(* CoDeSys 2.3.6.0 project: oscat13.pro *)
(* Libraries: SysLibRtc.lib 5.10.04 09:37:42, Standard.lib 22.11.04 11:21:12, SYSLIBCALLBACK.LIB 20.4.05 10:04:48, Util.lib 15.6.05 09:51:38 *)

(* PLC configuration (modules and I/O channels)
switch_1 AT %IX21.0 [BOOLOnX_I] Ch_1 Digital input
switch_2 AT %IX21.1 [BOOLOnX_I] Ch_2 Digital input
0750-0501 2 DO 24V DC 0.5A [Type_10_2_Channels] node 1, in %IB1 out %QB1 {INTTypePAAssignment = PLC; INTTypeModule = plugged}
  output_1 AT %QX19.0 [BOOLOnX_Q] Ch_1 Digital output
  output_2 AT %QX19.1 [BOOLOnX_Q] Ch_2 Digital output
0750-0501 2 DO 24V DC 0.5A [Type_10_2_Channels] node 2, in %IB2 out %QB2 {INTTypePAAssignment = PLC; INTTypeModule = plugged}
  output_3 AT %QX19.2 [BOOLOnX_Q] Ch_1 Digital output
  output_4 AT %QX19.3 [BOOLOnX_Q] Ch_2 Digital output
0750-0502 2 DO 24V DC 2.0A [Type_10_2_Channels] node 3, in %IB3 out %QB3 {INTTypePAAssignment = PLC; INTTypeModule = plugged}
  aus55 AT %QX19.4 [BOOLOnX_Q] Ch_1 Digital output
  AT %QX19.5 [BOOLOnX_Q] Ch_2 Digital output
0750-0501 2 DO 24V DC 0.5A [Type_10_2_Channels] node 4, in %IB4 out %QB4 {INTTypePAAssignment = PLC; INTTypeModule = plugged}
  heinz AT %QX19.6 [BOOLOnX_Q] Ch_1 Digital output
  AT %QX19.7 [BOOLOnX_Q] Ch_2 Digital output
0750-0523/0010-0000 1DO 230V AC 16A/Relay 1a/Potential free [Type_26_1_Channels] node 5, in %IB5 out %QB5 {INTTypePAAssignment = PLC; INTTypeModule = plugged}
  hand AT %IX21.2 [BOOLOnX_I] Diagnostic bit
  output_16A AT %QX19.8 [BOOLOnX_Q] Digital output
0750-0559 4 AO 0-10V DC [Type_14_4_Channels] node 6, in %IB6 out %QB6 {INTTypePAAssignment = PLC; INTTypeModule = plugged}
  AT %QW0 [WORDOnW_Q] Ch_1 Analog output
  AT %QW1 [WORDOnW_Q] Ch_2 Analog output
  AT %QW2 [WORDOnW_Q] Ch_3 Analog output
  AT %QW3 [WORDOnW_Q] Ch_4 Analog output
0750-0402 4 DI 24 V DC 3.0ms [Type_1_4_Channels] node 7, in %IB7 out %QB7 {INTTypePAAssignment = PLC; INTTypeModule = plugged}
  switch_3 AT %IX21.4 [BOOLOnX_I] Ch_1 Digital input
  switch_4 AT %IX21.5 [BOOLOnX_I] Ch_2 Digital input
  AT %IX21.6 [BOOLOnX_I] Ch_3 Digital input
  AT %IX21.7 [BOOLOnX_I] Ch_4 Digital input
0750-0402 4 DI 24 V DC 3.0ms [Type_1_4_Channels] node 8, in %IB8 out %QB8 {INTTypePAAssignment = PLC; INTTypeModule = plugged}
  AT %IX21.8 [BOOLOnX_I] Ch_1 Digital input
  AT %IX21.9 [BOOLOnX_I] Ch_2 Digital input
  AT %IX21.10 [BOOLOnX_I] Ch_3 Digital input
  AT %IX21.11 [BOOLOnX_I] Ch_4 Digital input
  AT %IX21.12 [BOOLOnX_I] Ch_1 Digital input
  AT %IX21.13 [BOOLOnX_I] Ch_2 Digital input
  AT %IX21.14 [BOOLOnX_I] Ch_3 Digital input
  AT %IX21.15 [BOOLOnX_I] Ch_4 Digital input
dcf77in AT %IX22.0 [BOOLOnX_I] Ch_1 Digital input
dcf77_2 AT %IX22.1 [BOOLOnX_I] Ch_2 Digital input
AT %IX22.2 [BOOLOnX_I] Ch_3 Digital input
AT %IX22.3 [BOOLOnX_I] Ch_4 Digital input
AT %IX22.4 [BOOLOnX_I] Ch_5 Digital input
AT %IX22.5 [BOOLOnX_I] Ch_6 Digital input
AT %IX22.6 [BOOLOnX_I] Ch_7 Digital input
AT %IX22.7 [BOOLOnX_I] Ch_8 Digital input
0750-0431 8 DI 24 V DC 0.2ms [Type_1_8_Channels] node 11, in %IB11 out %QB11 {INTTypePAAssignment = PLC; INTTypeModule = plugged}
  clkin AT %IX22.8 [BOOLOnX_I] Ch_1 Digital input
  AT %IX22.9 [BOOLOnX_I] Ch_2 Digital input
  AT %IX22.10 [BOOLOnX_I] Ch_3 Digital input
  AT %IX22.11 [BOOLOnX_I] Ch_4 Digital input
  AT %IX22.12 [BOOLOnX_I] Ch_5 Digital input
  AT %IX22.13 [BOOLOnX_I] Ch_6 Digital input
  AT %IX22.14 [BOOLOnX_I] Ch_7 Digital input
  AT %IX22.15 [BOOLOnX_I] Ch_8 Digital input
0750-0402 4 DI 24 V DC 3.0ms [Type_1_4_Channels] node 12, in %IB12 out %QB12 {INTTypePAAssignment = PLC; INTTypeModule = plugged}
  AT %IX23.0 [BOOLOnX_I] Ch_1 Digital input
  AT %IX23.1 [BOOLOnX_I] Ch_2 Digital input
  AT %IX23.2 [BOOLOnX_I] Ch_3 Digital input
  AT %IX23.3 [BOOLOnX_I] Ch_4 Digital input
0750-0531 4 DO 24V DC 0.5A [Type_10_4_Channels] node 13, in %IB13 out %QB13 {INTTypePAAssignment = PLC; INTTypeModule = plugged}
  AT %QX19.10 [BOOLOnX_Q] Ch_1 Digital output
  AT %QX19.11 [BOOLOnX_Q] Ch_2 Digital output
  AT %QX19.12 [BOOLOnX_Q] Ch_3 Digital output
  AT %QX19.13 [BOOLOnX_Q] Ch_4 Digital output
0750-0531 4 DO 24V DC 0.5A [Type_10_4_Channels] node 14, in %IB14 out %QB14 {INTTypePAAssignment = PLC; INTTypeModule = plugged}
  AT %QX19.14 [BOOLOnX_Q] Ch_1 Digital output
  AT %QX19.15 [BOOLOnX_Q] Ch_2 Digital output
  AT %QX20.0 [BOOLOnX_Q] Ch_3 Digital output
  AT %QX20.1 [BOOLOnX_Q] Ch_4 Digital output
0750-0531 4 DO 24V DC 0.5A [Type_10_4_Channels] node 15, in %IB15 out %QB15 {INTTypePAAssignment = PLC; INTTypeModule = plugged}
  AT %QX20.2 [BOOLOnX_Q] Ch_1 Digital output
  AT %QX20.3 [BOOLOnX_Q] Ch_2 Digital output
  AT %QX20.4 [BOOLOnX_Q] Ch_3 Digital output
  AT %QX20.5 [BOOLOnX_Q] Ch_4 Digital output
0750-0531 4 DO 24V DC 0.5A [Type_10_4_Channels] node 16, in %IB16 out %QB16 {INTTypePAAssignment = PLC; INTTypeModule = plugged}
  AT %QX20.6 [BOOLOnX_Q] Ch_1 Digital output
  AT %QX20.7 [BOOLOnX_Q] Ch_2 Digital output
  AT %QX20.8 [BOOLOnX_Q] Ch_3 Digital output
  AT %QX20.9 [BOOLOnX_Q] Ch_4 Digital output
0750-0504 4 DO 24V DC 0.5A [Type_10_4_Channels] node 17, in %IB17 out %QB17 {INTTypePAAssignment = PLC; INTTypeModule = plugged}
  AT %QX20.10 [BOOLOnX_Q] Ch_1 Digital output
  AT %QX20.11 [BOOLOnX_Q] Ch_2 Digital output
  AT %QX20.12 [BOOLOnX_Q] Ch_3 Digital output
  AT %QX20.13 [BOOLOnX_Q] Ch_4 Digital output
0750-0550 2 AO 0-10V DC [Type_14_2_Channels] node 18, in %IB18 out %QB18 {INTTypePAAssignment = PLC; INTTypeModule = plugged}
  aout1 AT %QW4 [WORDOnW_Q] Ch_1 Analog output
  AT %QW5 [WORDOnW_Q] Ch_2 Analog output
0750-0556 2 AO ±10V [Type_14_2_Channels] node 19, in %IB19 out %QB19 {INTTypePAAssignment = PLC; INTTypeModule = plugged}
  AT %QW6 [WORDOnW_Q] Ch_1 Analog output
  AT %QW7 [WORDOnW_Q] Ch_2 Analog output
0750-0654 DataExchange Module [Type_23_1_Channels] node 20, in %IB20 out %QB20 {INTTypePAAssignment = PLC; INTTypeModule = plugged}
  AT %IX0.0 [BOOLOnX_I] Parity error or wrong data in a frame
  AT %IX0.1 [BOOLOnX_I] Buffer overflow
  AT %IX0.2 [BOOLOnX_I] Checksum error
  AT %IX0.3 [BOOLOnX_I] receiver timeout
  AT %IX0.4 [BOOLOnX_I] Module timeout
  AT %IB1 [BYTEOnB_I] Input data Byte 0
  AT %IB2 [BYTEOnB_I] Input data Byte 1
  AT %IB3 [BYTEOnB_I] Input data Byte 2
  AT %QB17 [BYTEOnB_Q] Output data Byte 0
  AT %QB18 [BYTEOnB_Q] Output data Byte 1
  AT %QB19 [BYTEOnB_Q] Output data Byte 2
0750-0460 4 AI PT100 (RTD) [Type_44_4_Channels] node 21, in %IB21 out %QB21 {INTTypePAAssignment = PLC; INTTypeModule = plugged}
  AT %IW2 [INTOnW_I] Ch_1 signed Input value
  AT %IW3 [INTOnW_I] Ch_2 signed Input value
  AT %IW4 [INTOnW_I] Ch_3 signed Input value
  AT %IW5 [INTOnW_I] Ch_4 signed Input value
0750-0454 2 AI 4-20mA Diff [Type_8_2_Channels] node 22, in %IB22 out %QB22 {INTTypePAAssignment = PLC; INTTypeModule = plugged}
  AT %IW6 [WORDOnW_I] Ch_1 Input word
  AT %IW7 [WORDOnW_I] Ch_2 Input word
  Ain1 AT %IW8 [WORDOnW_I] Ch_1 Input word
  Ain2 AT %IW9 [WORDOnW_I] Ch_2 Input word
0750-0550 2 AO 0-10V DC [Type_14_2_Channels] node 24, in %IB24 out %QB24 {INTTypePAAssignment = PLC; INTTypeModule = plugged}
  AT %QW10 [WORDOnW_Q] Ch_1 Analog output
  AT %QW11 [WORDOnW_Q] Ch_2 Analog output
0750-0650 RS 232 C Interface (9600/8/1/N) [Type_21_1_Channels] node 25, in %IB25 out %QB25 {INTTypePAAssignment = PLC; INTTypeModule = plugged}
  AT %IX10.0 [BOOLOnX_I] Transmission acknowledgement
  AT %IX10.1 [BOOLOnX_I] Reception request
  AT %IX10.2 [BOOLOnX_I] Initialization acknowledgement
  AT %IX10.3 [BOOLOnX_I] Input buffer is full
  AT %IX10.4 [BOOLOnX_I] Number of received characters Bit 0
  AT %IX10.5 [BOOLOnX_I] Number of received characters Bit 1
  AT %IX10.6 [BOOLOnX_I] Number of received characters Bit 2
  AT %IB21 [BYTEOnB_I] Input data Byte 0
  AT %IB22 [BYTEOnB_I] Input data Byte 1
  AT %IB23 [BYTEOnB_I] Input data Byte 2
  AT %QX12.0 [BOOLOnX_Q] Transmission request
  AT %QX12.1 [BOOLOnX_Q] Reception acknowledgement
  AT %QX12.2 [BOOLOnX_Q] Initialization request
  AT %QX12.4 [BOOLOnX_Q] Number of characters Bit 0
  AT %QX12.5 [BOOLOnX_Q] Number of characters Bit 1
  AT %QX12.6 [BOOLOnX_Q] Number of characters Bit 2
  AT %QB25 [BYTEOnB_Q] Output data Byte 0
  AT %QB26 [BYTEOnB_Q] Output data Byte 1
  AT %QB27 [BYTEOnB_Q] Output data Byte 2
0750-0641 DALI/DSI-Master [Type_36_1_Channels] node 26, in %IB26 out %QB26 {INTTypePAAssignment = PLC; INTTypeModule = plugged}
  AT %IX12.0 [BOOLOnX_I] Transmit accepted
  AT %IX12.1 [BOOLOnX_I] Receive request
  AT %IX12.2 [BOOLOnX_I] Init accepted
  AT %IX12.3 [BOOLOnX_I] Actor Error
  AT %IX12.4 [BOOLOnX_I] Frame Error
  AT %IX12.5 [BOOLOnX_I] Bus Error
  AT %IX12.6 [BOOLOnX_I] General Module Error
  AT %IB25 [BYTEOnB_I] DALI Response
  AT %IB26 [BYTEOnB_I] DALI Address
  AT %IB27 [BYTEOnB_I] Message 3
  AT %IB28 [BYTEOnB_I] Message 2
  AT %IB29 [BYTEOnB_I] Message 1
  AT %QX14.0 [BOOLOnX_Q] Transmit request
  AT %QX14.1 [BOOLOnX_Q] Receive accepted
  AT %QX14.2 [BOOLOnX_Q] Init request
  AT %QB29 [BYTEOnB_Q] DALI Command, DSI dimming value
  AT %QB30 [BYTEOnB_Q] DALI Address
  AT %QB31 [BYTEOnB_Q] Parameter 2
  AT %QB32 [BYTEOnB_Q] Parameter 1
  AT %QB33 [BYTEOnB_Q] Command extension
0750-0460 4 AI PT100 (RTD) [Type_44_4_Channels] node 27, in %IB27 out %QB27 {INTTypePAAssignment = PLC; INTTypeModule = plugged}
  AT %IW15 [INTOnW_I] Ch_1 signed Input value
  AT %IW16 [INTOnW_I] Ch_2 signed Input value
  AT %IW17 [INTOnW_I] Ch_3 signed Input value
  AT %IW18 [INTOnW_I] Ch_4 signed Input value
0750-0642 EnOcean/RF-Receiver [Type_37_1_Channels] node 28, in %IB28 out %QB28 {INTTypePAAssignment = PLC; INTTypeModule = plugged}
  AT %IX19.0 [BOOLOnX_I] Transmission acknowledgement
  AT %IX19.1 [BOOLOnX_I] Reception request
  AT %IX19.2 [BOOLOnX_I] Initialization acknowledgement
  AT %IX19.3 [BOOLOnX_I] Number of received characters Bit 0
  AT %IX19.4 [BOOLOnX_I] Number of received characters Bit 1
  AT %IX19.5 [BOOLOnX_I] Number of received characters Bit 2
  AT %IX19.6 [BOOLOnX_I] Input buffer is full
  AT %IB39 [BYTEOnB_I] Input data Byte 0
  AT %IB40 [BYTEOnB_I] Input data Byte 1
  AT %IB41 [BYTEOnB_I] Input data Byte 2
  AT %QX17.0 [BOOLOnX_Q] Transmission request
  AT %QX17.1 [BOOLOnX_Q] Reception acknowledgement
  AT %QX17.2 [BOOLOnX_Q] Initialization request
0750-0517 2 DO 230V AC 1.0A Rel 2CO (PotFree) [Type_10_2_Channels] node 29, in %IB29 out %QB29 {INTTypePAAssignment = PLC; INTTypeModule = plugged}
  AT %QX20.14 [BOOLOnX_Q] Ch_1 Digital output
  AT %QX20.15 [BOOLOnX_Q] Ch_2 Digital output
0750-0517 2 DO 230V AC 1.0A Rel 2CO (PotFree) [Type_10_2_Channels] node 30, in %IB30 out %QB30 {INTTypePAAssignment = PLC; INTTypeModule = plugged}
  AT %QX21.0 [BOOLOnX_Q] Ch_1 Digital output
  AT %QX21.1 [BOOLOnX_Q] Ch_2 Digital output
win_o AT %IX256.0 [BOOLOnX_I] BOOL
wout_i AT %QX256.0 [BOOLOnX_Q] BOOL
*)

(* Global variable list: Constants *)
VAR_GLOBAL CONSTANT
	PI : REAL := 3.14159265358979323846264338327950288;
	PI2 : REAL := 6.283185307;
	e : REAL := 2.71828182845904523536028747135266249;
END_VAR

VAR_GLOBAL
	ontime: TIME;
END_VAR

(* Global variable list: Globale_Variablen *)
VAR_GLOBAL

	(* 	time and date variables		*)
	gmt : DT;						(*	world time				*)
	DST_enable : BOOL;					(* 	daylight saving time active	*)
	localtime : DT;				(*	current local time			*)
	sun_offset : TIME;				(*	offset of astrological midday in hours when sun stand at south direction	*)
	sun_rise : TOD;				(*	sun rise for current day in local time *)
	sun_set : TOD;				(*	sun set for current day in local time *)
	sun_declination : REAL;		(*	sun angle at midday	*)

	(*	environmental data			*)
	external_temperature : REAL;	(*	outside temperature in °C	*)
	wind_speed : REAL;			(*	wind speed in km/h			*)

END_VAR

(* Global variable list: Setup_Data *)
VAR_GLOBAL RETAIN

(*	geographical position		*)
	latitude : REAL;		(*	geographical position in degrees north of equator			*)
	longitude : REAL;		(*	geographical position in degrees east of prime meridian		*)
	elevation : REAL;		(*	elevation												*)

(*	time zone data			*)
	Time_zone_offset : TIME;		(*	local time zone offset		*)

END_VAR

(* POU mathematical/array functions/_array_init, ST *)
FUNCTION _array_init : REAL
VAR_INPUT
	pt : POINTER TO ARRAY[0..32000] OF REAL;
	size : INT;
	init : REAL;
END_VAR
VAR
	i: INT;
	stop: INT;
END_VAR


(*
version 1.0	2 oct 2006
programmer 	hugo
tested by		tobias

this function will initialize a given array with a value init.
the function needs to be called:	_array_init(adr("array"),sizeof("array"));
this function will manipulate a given array.
the function will not return anything, it will instead manipulate the original array.
because this function works with pointers its very time efficient and it needs no extra memory.

*)
stop := (size - SIZEOF(pt)) / SIZEOF(pt);
FOR i := 0 TO stop DO
	pt^[i] := init;
END_FOR;
END_FUNCTION

(* POU mathematical/array functions/_array_median, ST *)
FUNCTION _array_median : REAL
VAR_INPUT
	pt : POINTER TO ARRAY[0..32000] OF REAL;
	size : INT;
END_VAR
VAR
	i: INT;
	m: INT;
	temp : REAL;
	stop: INT;
END_VAR

(*
version 1.0	2 oct 2006
programmer 	hugo
tested by		tobias

this function will calculate the median of a given array.
in order to do so the ariginal array is sorted and stays sorted after the function finishes
the function needs to be called:	_array_median(adr("array"),sizeof("array"));
this function will manipulate a given array.
the function will return the median of the original array.
for example [12,0,4,7,1] the median is 4 and the array after the function is called is [0,1,4,7,12]
because this function works with pointers its very time efficient and it needs no extra memory.

*)
stop := (size - SIZEOF(pt)) / SIZEOF(pt);
FOR i := 0 TO stop - 1 DO
	FOR m := i + 1 TO stop DO
		IF pt^[i] > pt^[m] THEN
			temp := pt^[i];
			pt^[i] := pt^[m];
			pt^[m] := temp;
		END_IF;
	END_FOR;
END_FOR;
IF even(stop) THEN
	_array_median := pt^[stop/2];
ELSE
	i := TRUNC(stop/2);
	_array_median := (pt^[i] + pt^[i+1])/2;
END_IF;
END_FUNCTION

(* POU mathematical/even, ST *)
FUNCTION even : BOOL
VAR_INPUT
	in : INT;
END_VAR
VAR
	test: INT;
END_VAR


(*
version 1.0	1 oct 2006
programmer 	hugo
tested by		tobias

this function chacks an input for even  value
the output is true if the input is even.
execution time on wago 750 - 841 =  10  us
*)
IF (in MOD 2) = 0 THEN  even := TRUE; ELSE even := FALSE; END_IF;
END_FUNCTION

(* POU mathematical/array functions/_array_sort, ST *)
FUNCTION _array_sort : BOOL
VAR_INPUT
	pt : POINTER TO ARRAY[0..32000] OF REAL;
	size : INT;
END_VAR
VAR
	i: INT;
	m: INT;
	temp : REAL;
	stop: INT;
END_VAR

(*
version 1.0	2 oct 2006
programmer 	hugo
tested by		tobias

this function will sort a given array.
the function needs to be called:	_array_sort(adr("array"),sizeof("array"));
this function will manipulate a given array.
the function will not return anything, it will instead manipulate the original array.
because this function works with pointers its very time efficient and it needs no extra memory.

*)
stop := (size - SIZEOF(pt)) / SIZEOF(pt);
FOR i := 0 TO stop - 1 DO
	FOR m := i + 1 TO stop DO
		IF pt^[i] > pt^[m] THEN
			temp := pt^[i];
			pt^[i] := pt^[m];
			pt^[m] := temp;
		END_IF;
	END_FOR;
END_FOR;
_array_sort := FALSE;
END_FUNCTION

(* POU Building/HLK/actuator_2P, ST *)
FUNCTION_BLOCK actuator_2P
VAR_INPUT
	val : REAL;
	force : BOOL;
	force_in : BOOL;
END_VAR
VAR_INPUT CONSTANT
	self_act_time : TIME := t#10d;
	self_act_cycles : INT := 5;
	cycle_time : TIME := t#10m;
	min_ontime : TIME := t#10s;
	min_offtime : TIME := t#10s;
END_VAR
VAR_OUTPUT
	out :BOOL;
	pos : REAL;
END_VAR
VAR
	last_activation : TIME;
	time_overflow : BOOL;
	count : INT;
	TON : TIME;
END_VAR


(*
version 1.1	7 oct 2006
programmer 	hugo
tested by		tobias

this is an intelligent actuator interface for any 2point actuator like coil drive.
the 2Point actuator can only switch on/off and therefore a input must be converted to on/off cycles.
the interface can be programmed with double click on the symbol for duty cyle, min_ontime and min_offtime to avoid flickering of the valve or flap.
in addition a self_act_time and self_act_cycles ca be programmed to switch n times on/off every self_act_time to avoid a valve to freeze.
a on and off input can be used to force the valve on or off at all times.
a additional pos output will always indicate the current position of a valve.
the input value must be between 0 and 1.

val		force	force_in	pos	out			
X		0		-			X		duty cycle X
-		1		1			1		1
-		1		0			0		0

*)
(* verify input to be between 0 and 1 *)
IF val <0 THEN val := 0; ELSIF val > 1 THEN val := 1; END_IF;

(* check for min ontime or min offtime and wait if not passed *)
IF (out AND TIME() - last_activation < min_ontime) OR (NOT out AND TIME() - last_activation < min_offtime) THEN RETURN;

(* when force off then shutoff valve *)
ELSIF force AND NOT force_in THEN
	pos := 0;
	out := 0;
	last_activation := TIME();
	count := 0;

(* if force on then turn on valve *)

ELSIF force AND force_in THEN
	pos := 1;
	out := 1;
	last_activation := TIME();
	count := 0;

(* if nothing happened for self_act_time then do self activation cycles *)
ELSIF (TIME() - last_activation >= self_act_time AND count = 0 AND self_act_cycles > 0) OR (count > 0 AND count < self_act_cycles * 2) THEN
	out := NOT out;
	last_activation := TIME();
	count := count + 1;
	RETURN;
ELSIF count > 0 THEN
	count := 0;
ELSE
	ton := multime(cycle_time,val);
	IF ton < min_ontime / 2 THEN ton := t#0s; ELSIF ton < min_ontime THEN ton := min_ontime; END_IF;
	IF ton > cycle_time - min_offtime / 2 THEN ton := cycle_time; ELSIF ton > cycle_time - min_offtime THEN ton := cycle_time - min_offtime; END_IF;
	IF ton = t#0s THEN
		IF out =0 THEN
			pos := 0;
			RETURN;
		ELSE
			out := 0;
			pos := 0;
			last_activation := TIME();
		END_IF;
	ELSIF ton = cycle_time THEN
		IF out = 1 THEN
			pos := 1;
			RETURN;
		ELSE
			out := 1;
			pos := 1;
			last_activation := TIME();
		END_IF;
	END_IF;
	pos := TIME_TO_REAL(ton) / TIME_TO_REAL(cycle_time);
	(* output pulse generation *)
	IF out AND TIME() - last_activation >= ton THEN
		out := 0;
		last_activation := TIME();
	ELSIF NOT out AND TIME() - last_activation >= cycle_time - ton THEN
		out := 1;
		last_activation := TIME();
	END_IF;
END_IF;


(*
revision history:

7.10.2006: changes on and off in the be force and force_in for better usability.
7.10.2006: changed error pos could not reach 1 or 0 under certain conditions due to error in code.

*)
END_FUNCTION_BLOCK

(* POU engineering/measurements/cycle_time, ST *)
FUNCTION_BLOCK cycle_time
VAR_INPUT
	rst : BOOL;
END_VAR
VAR_OUTPUT
	ct_min : TIME := t#0s;
	ct_max : TIME := t#0s;
	ct_last : TIME;
	systime : TIME;
	sysdays : INT;
	cycles : DWORD;
END_VAR
VAR
	last_cycle : TIME;
	tx: TIME;
	init: BOOL;
END_VAR


(*
	version 1.1	12 dec 2006
	programmer 	hugo
	tested BY		hans

this function block measures the cycle time and displays the last, min and max cycle time of the current task.
the resolution is 1ms.
the cycles output is a dword counter which counts the cycles.
a rst pulse on the input will reset all data.


*)
tx :=TIME() - last_cycle;
IF rst THEN
	ct_min := t#0s - t#1ms;
	ct_max := t#0ms;
	cycles := 0;
ELSIF last_cycle > t#0s THEN
	IF tx < ct_min THEN ct_min := tx;
	ELSIF tx > ct_max THEN ct_max := tx;
	END_IF;
	ct_last := tx;
ELSIF ct_min = t#0s THEN
	ct_min := t#0s - t#1ms;
END_IF;
IF init THEN
	systime := systime + tx;
		IF systime >= t#1d THEN
			systime := systime - t#1d;
			sysdays := sysdays + 1;
		END_IF;
END_IF;
init := TRUE;
last_cycle := last_cycle + tx;
cycles := cycles + 1;

(* hm 12.12.2006		rev 1.1

added cycles output, a dword cycle counter.

*)
END_FUNCTION_BLOCK

(* POU Time&Date/multime, ST *)
FUNCTION multime : TIME
VAR_INPUT
	t : TIME;
	M : REAL;
END_VAR
VAR
END_VAR


(*
version 1.0	2 oct 2006
programmer 	hugo
tested by		tobias

multiplies a time by a real number and returns a time
*)
multime := REAL_TO_TIME(TIME_TO_REAL(t)*M);
END_FUNCTION

(* POU Building/HLK/actuator_3P, ST *)
FUNCTION_BLOCK actuator_3P
VAR_INPUT
	in : REAL;
	force : BOOL;
	on : BOOL;
	end_pos : BOOL;
	diag : BOOL;
END_VAR
VAR_INPUT CONSTANT
	min_ontime : TIME := t#10s;
	min_offtime : TIME := t#10s;
	max_runtime : TIME := t#60s;
	auto_diag_time : TIME := t#10d;
	cal_runtime : TIME := t#600s;
	switch_available: BOOL;
END_VAR
VAR_OUTPUT
	out1 : BOOL;
	out2 : BOOL;
	pos : REAL;
	busy : BOOL;
	error : BOOL;
END_VAR
VAR
	val: REAL;
	tx : TIME;
	last_diag: TIME;
	last : TIME;
	runtime_1 : TIME;
	runtime_2 : TIME;
	state : INT;
	force_on : BOOL;
	force_off : BOOL;
	rout: FT_rmp;
	end : R_TRIG;
	cal_timer: TIME;
END_VAR


(*
version 1.1	19 oct 2006
programmer 	hugo
tested by		tobias

actuator_3P is an interface for a 3 point actuator.
a 3P actuator is a motor with 2 directions that drives a valve or flap. the position of the valve or flap is controlled by runtime of the motor foreward or backward.
the available inputs are:
in is a real value which specifies the position of the actuator, 0 = 0% and 1 = 100% any value <0 or > 1 is limited to 0 or 1.
a force input must be low for normal operation and if switched high, the motor can only be controlled for 0% or 100% positions with the on input.
an and pos input is available for a end_pos switch, this switch indicates the valve or flap to be at either 0% or 100%
a diag input can at any time start a diag cycle which turns the motor towards the 0% position, then measures the runtime to 100% and then the runtime to 0%
these runtimes are stored and used for absolute positioning of the motor during normal operation.
a setup constand "auto_diag_time can be used to specify how often the actuator repeates this auto_diag cycla automatically.
at power on a cycle is perfomed automatically.
a 0 for this value means auto diag is never performed.

the outputs ar out1 and out2 for up and down direction of the motor. to avoid flickering the output can be programmed for min_ontime and min_offtime.
a pos outout indicates the absulute position of the actuator during operation and a busy output indicates the actuator is busy.
a error output is initiated when the specified max_runtime is reached by any direction during debug.
also when the up and down direction differs by more then 10% the error output is set.

for absolute positioning accuracy the actuator has a setup variable "cal_runtime" if this is set the actuator measures the total runtime of the motors and when this 
cal_runtime is exceeded it resets the actuator to 0% position and sets the output again to assure absolute accuracy.

autodiag and calibration can be shut off by setting the appropriate values to 0.
a switch_available setup variable specifies if end_pos switches are available.

*)
(* setup *)
tx := TIME() - last;
end(clk := end_pos);

(* init only when first started *)
IF state = 0 THEN
	runtime_1 := max_runtime;
	runtime_2 := max_runtime;
	state := 1;
	rout(KR := 1000 / TIME_TO_REAL(runtime_1), KF := 1000 / TIME_TO_REAL(runtime_1) );
	tx := t#0s;
	last := TIME();
	last_diag := last;
END_IF;

(* check for end_sw and stop if reached *)
IF switch_available AND out1 AND end.Q THEN
	(* upper limit has been reached *)
	out1 := 0;
	rout(rmp := 0, in := 1);
	rout.Rmp := 1;
ELSIF switch_available AND out2 AND end.Q THEN
	(* lower limit has been reached *)
	out2 := 0;
	rout(rmp := 0, in := 0);
	rout.Rmp := 1;
END_IF;

(* check for min_offtime and min_ontime and return if it has not elapsed *)
IF NOT busy AND tx < min_offtime THEN RETURN;
ELSIF busy AND tx < min_ontime THEN RETURN;

(* check for last diag cycle and start diag if auto_diag_time has elapsed *)
ELSIF (tx + last - last_diag > auto_diag_time AND state > 10 AND auto_diag_time > t#0s) OR (diag AND state >= 10) THEN state := 1;

(* check if force pin is high *)
ELSIF force THEN state := 10;

(* check if calibration is necessary *)
ELSIF cal_timer > cal_runtime AND state = 99 AND cal_runtime > t#0s THEN state := 20;
END_IF;

(* state machine for operation *)
CASE state OF

1 :	(* diagnostic start *)
	(* all data is reset and out2 is turned on to make sure we start from top position *)
	last_diag := tx + last;
	diag := 0;
	state := 2;
	pos := 0;
	busy := 1;
	last := tx + last;
	out1 := 0;
	out2 := 1;
	RETURN;

2:	(* wait for max_runtime or end_pos to be reached *)
	IF tx < max_runtime AND NOT end.Q THEN RETURN; END_IF;
	state := 3;
	last := tx + last;
	out1 := 1;
	out2 := 0;
	RETURN;

3: 	(* measure runtime_2 *)
	IF tx < max_runtime AND NOT end.Q THEN RETURN; END_IF;
	state := 4;
	runtime_1 := tx;
	last := tx + last;
	out1 := 0;
	out2 := 1;
	RETURN;

4:	(* measure runtime_1 *)
	IF tx < max_runtime AND NOT end.Q THEN RETURN; END_IF;
	state := 99;
	runtime_2 := tx;
	last := tx + last;
	out2 := 0;
	busy := 0;
	(* reset the output ramp generator to the 0% position as the valve is after diags *)
	rout(rmp := 0, in := 0);
	rout.Rmp := 1;
	cal_timer := t#0s;
	IF differ(TIME_TO_REAL(runtime_1), TIME_TO_REAL(runtime_2), TIME_TO_REAL(max_runtime) * 0.1) THEN error := TRUE;
	ELSIF runtime_1 > multime(max_runtime, 0.9) AND switch_available THEN error := TRUE;
	ELSIF runtime_2 > multime(max_runtime, 0.9) AND switch_available THEN error := TRUE;
	END_IF;
	RETURN;

10: (* force pin is active, outputs are forced on or off by the on pin *)
	IF on AND NOT out2 THEN val := 1;
	ELSIF NOT on AND NOT out1 THEN val := 0;
	END_IF;
	IF NOT force THEN state := 99; END_IF;

20 : (* calibrate to allow for correction of positioning error addig up *)
	cal_timer := t#0s;
	state := 21;
	pos := 0;
	busy := 1;
	last := tx + last;
	out1 := 0;
	out2 := 1;
	RETURN;

21:	(* after end_sw or max_runtime we can be sure to have reached the 0% position *)
	IF tx < max_runtime AND NOT end.Q THEN RETURN; END_IF;
	state := 99;
	out2 := 0;
	busy := 0;
	last := tx + last;
	rout(rmp := 0, in := 0);
	rout.Rmp := 1;
	RETURN;

99: (* normal operation *)
	(* only if input changes for an equivalent of min_ontime then change the output *)
	(* if there is a directional change then wait until last step is finished *)
	IF in < TIME_TO_REAL(min_ontime)/TIME_TO_REAL(max_runtime)/2 THEN val := 0;
	ELSIF in > 1 - TIME_TO_REAL(min_ontime)/TIME_TO_REAL(max_runtime)/2 THEN val := 1;
	ELSIF differ(LIMIT(0,in,1), val, TIME_TO_REAL(min_ontime) / TIME_TO_REAL(max_runtime)) OR in = 0 OR in = 1 THEN
		IF in < val AND NOT out1 THEN val := in;
		ELSIF in > val AND NOT out2 THEN val := in;
		END_IF;
	END_IF;

END_CASE;

(* output ramp generator *)
rout(in := val);
out1 := rout.busy AND rout.UD;
out2 := rout.busy AND NOT rout.UD;
pos := rout.out;

(* set the busy output and if busy goes low, then set the last time in order to check for min_offtime *)
IF NOT busy AND rout.busy THEN
	last := tx + last;
ELSIF busy AND NOT rout.busy THEN
	cal_timer := cal_timer + tx;
	last := tx + last;
END_IF;
busy := rout.busy;



(* revision history

19.10.2006	added security checks for end_switch to avoid overrun of the end_switch, hans

*)
END_FUNCTION_BLOCK

(* POU mathematical/functions/FT_rmp, ST *)
FUNCTION_BLOCK FT_rmp
VAR_INPUT
	Rmp : BOOL := TRUE;
	in : REAL;
	KR : REAL;
	KF : REAL;
END_VAR
VAR_OUTPUT
	out : REAL;
	busy : BOOL;
	UD : BOOL;
END_VAR
VAR
	tx: TIME;
	last: TIME;
END_VAR

(*
	version 1.1	8 oct 2006
	programmer 	oscat
	tested BY		oscat

this ramp function follows an input signal with a linear ramp up or down, the up or down speed can be set with KF and KR.
a K factor of 1 means 1 unit per second on the output. K factors can only be positive and not negative.
a busy output signals the ramp is running or busy false means the in value is present on the output.
a rmp input false means the output follows the input dierctly while a rmp = true means the output follows the input with a ramp.
a updn output signal the directon of the ramp (up or down).

*)
tx := TIME() - last;
IF NOT rmp THEN
	out := in;
	busy := FALSE;
ELSIF out > in AND kf > 0 THEN
	(* ramp down *)
	out := out - TIME_TO_REAL(tx) / 1000 * KF;
	IF out < in THEN out := in; END_IF;
ELSIF out < in AND kr > 0 THEN
	(* ramp up *)
	out := out + TIME_TO_REAL(tx) / 1000 * KR;
	IF out > in THEN out := in; END_IF;
END_IF;

(* set busy and dir flags *)
IF out < in THEN
	busy := TRUE;
	ud := 1;
ELSIF out > in THEN
	busy := TRUE;
	ud := 0;
ELSE
	busy := FALSE;
END_IF;
last := last + tx;


(* revision history:

8.10.2006		added ud output

*)
END_FUNCTION_BLOCK

(* POU mathematical/differ, ST *)
FUNCTION differ : BOOL
VAR_INPUT
	in1 : REAL;
	in2 : REAL;
	X : REAL;
END_VAR
VAR
END_VAR

(*
version 1.0	8 oct 2006
programmer 	hugo
tested by		tobias

this function checks if in1 differs more then x from in2
the output is true if in1 < in2 - x or in1 > in2 + X
*)
differ := in1 < in2 - X OR in1 > in2 + X;
END_FUNCTION

(* POU Building/actuator_pump, ST *)
FUNCTION_BLOCK actuator_pump
VAR_INPUT
	in : BOOL;
	manual : BOOL;
	rst : BOOL := FALSE;
END_VAR
VAR_INPUT CONSTANT
	min_ontime : TIME := t#10s;
	min_offtime : TIME := t#10s;
	run_every : TIME := t#10000m;
END_VAR
VAR_OUTPUT
	pump : BOOL;
	runtime : REAL;
	cycles : REAL;
END_VAR
VAR
	tx : TIME;
	last_change : TIME;
	meter : ontime;
	old_man : BOOL;
END_VAR

(*
	version 1.0	4 dec 2006
	programmer 	oscat
	tested BY		oscat

actuator_pump is a pump interface which cam be controlled by an input in and an input manual.
in or manual high turns the pump output on.
a rst input is used to reset the runtime counters.
when the pump was not active for a time run_every the actuator turns on the pump automatically for min_ontime.
two setup variables min_ontime and min_offtime guarantee a minimum runtime and offtime of the pump.
the units are hours and the output type is real to prevent fromoverfow.

*)
tx := TIME();
IF rst THEN
	rst := FALSE;
	meter(rst := 1);
	meter.rst := 0;
ELSIF manual AND NOT pump AND NOT old_man THEN
	last_change := tx;
	pump := 1;
ELSIF NOT manual AND old_man AND pump AND NOT in THEN
	last_change := tx;
	pump := 0;
ELSIF in AND NOT pump AND tx - last_change >= min_offtime THEN
	last_change := tx;
	pump := 1;
ELSIF pump AND NOT in AND NOT manual AND tx - last_change >= min_ontime THEN
	last_change := tx;
	pump := 0;
ELSIF NOT pump AND tx - last_change >= run_every THEN
	last_change := tx;
	pump := 1;
END_IF;

meter(in := pump);
runtime := meter.ontime;
cycles := meter.cycles;
old_man := manual;
END_FUNCTION_BLOCK

(* POU engineering/measurements/ontime, ST *)
FUNCTION_BLOCK ontime
VAR_INPUT
	in : BOOL;
	rst : BOOL := FALSE;
END_VAR
VAR_OUTPUT RETAIN PERSISTENT
	ontime : REAL;
	last_on : REAL;
	cycles : REAL;
END_VAR
VAR
	tx: TIME;
	last : TIME;
	power : BOOL := FALSE;
	edge : BOOL := 0;
END_VAR

(*
version 1.0	4 aug 2006
programmer 	oscat
tested by		tobias

M_runtime measures the ontime of a signal in hours.
the output is of type real because the time type will overflow within 49 days.
the units are hours.

*)
(* at first we need to determine if the sps was powered off *)

tx := TIME();
IF NOT power THEN
	power := TRUE;
	cycles := cycles +1;
ELSIF rst THEN
	ontime := 0;
	cycles := 0;
	last_on := 0;
ELSIF in THEN
	ontime := ontime + DWORD_TO_REAL( TIME_TO_DWORD(tx - last))/3600000.0;
	last_on := last_on + DWORD_TO_REAL(TIME_TO_DWORD(tx - last))/3600000.0;
	IF in AND NOT edge THEN
		cycles := cycles +1;
		last_on := 0;
	END_IF;
END_IF;
last := tx;
edge := in;
END_FUNCTION_BLOCK

(* POU Building/actuator_UD, ST *)
FUNCTION_BLOCK actuator_UD
VAR_INPUT
	UD : BOOL;
	ON : BOOL;
	TON : TIME;
	TOF : TIME;
	Manual : BOOL := 0;
	Up : BOOL;
	Dn : BOOL;
	off : BOOL := 0;
	YUP_in : BOOL;
	YDN_in : BOOL;
END_VAR

VAR_OUTPUT
	Yup : BOOL;
	Ydn : BOOL;
END_VAR
VAR
	tx : TIME;
	last : TIME;
	init: BOOL;
END_VAR

(*
version 1.0	12 Nov 2006
programmer 	hugo
tested by		tobias

out_ud is a up/dn or Right/left locked output driver.
if can be controlled by automatic inputs UD and ON as well as manual inputs for up and dn.
a security input to shut off at any time is prvided by the off input.
to time set inputs ton and toff specify a minimum on time for outputs and a minimum off time befoore the next output can become active.
the module assures that only one output can be active at any time.
for higher security pls make sure you use hardware locking of the outputs to prevent from defective wiring or outputs.
further security is provided b feedback inputs Yup_in and Ydn_in which are separate inputs for the output signal, if these inputs are not available 
pls connect them directly to Yup and Ydn.
automatic mode can override manual mode by setting the on input high while the manual input is high.

*)
tx := TIME();
IF NOT init THEN
	(* INITIALIZATION AT FIRST CALL *)
	last := tx;
	init := TRUE;
ELSIF off THEN
	(* emergency shut off detected *)
	Yup := FALSE;
	Ydn := FALSE;
	last := tx;
ELSIF ((Yup OR Ydn) AND tx - last < Ton) OR ((NOT Yup AND NOT Ydn) AND tx - last < tof) THEN
	(* WATH FOR MIN TON AND TOF TIME *)
	RETURN;
ELSIF manual AND NOT on THEN
	(* manual operation detected *)
	IF UP AND NOT DN AND NOT OFF THEN
		Ydn := 0;
		IF NOT Ydn_in THEN Yup := 1; END_IF;
		last := tx;
	ELSIF DN AND NOT UP AND NOT OFF THEN
		Yup := 0;
		IF NOT Yup_in THEN Ydn := 1; END_IF;
		last := tx;
	ELSE
		IF YUP OR YDN THEN LAST := tx; END_IF;
		Yup := 0;
		Ydn := 0;
	END_IF;
ELSE
	(* automatic operation *)
	IF Ud AND on AND NOT OFF THEN
		Ydn := 0;
		IF NOT ydn_in THEN Yup := 1; END_IF;
		last := tx;
	ELSIF NOT UD AND on AND NOT OFF THEN
		Yup := 0;
		IF NOT yup_in THEN Ydn := 1; END_IF;
		last := tx;
	ELSE
		IF Yup OR Ydn THEN last := tx; END_IF;
		Yup := 0;
		Ydn := 0;
	END_IF;
END_IF;

(* make sure Yup and Ydn are never on at the same time *)
IF Ydn AND Yup_in THEN Ydn := 0; END_IF;
IF Yup AND Ydn_in THEN Yup := 0; END_IF;
END_FUNCTION_BLOCK

(* POU engineering/signal conditioning/AIN, ST *)
FUNCTION AIN : REAL
VAR_INPUT
	in : DWORD;
END_VAR
VAR_INPUT CONSTANT
	Bits : BYTE;
	sign : BYTE := 255;
	low : REAL := 0;
	high : REAL := 10;
END_VAR
VAR
	temp1 : DWORD;
	temp2 : DWORD;
	sx : BOOL;
END_VAR

(*
version 1.1	18 aug 2006
programmer 	oscat
tested by		tobias

Ain converts signals from A/D converters or other analog sources to an internal real value
the lowest number of bits are extracted from the input word and the sign will be extracted if available separately.
the output signal is then conditioned to range from low to high values for a 0 to max value on the analog inputs:
for example a 15bit input (bits := 12) with sign at bit 15 (0..15) will deliver 0.0 (low value at 0) for an input value of 2#0000_0000_0000
an input value of 2#1111_1111_1111 will deliver 10.0 on the output (high value set to 10).

*) 
(* extract the sign bit *)
IF sign < 32 THEN
	temp1 := SHR(in,sign);
	sx := temp1.0;
ELSE
	sx := FALSE;
END_IF;
temp1 := SHR(16#FFFFFFFF,32-bits);
temp2 := in AND temp1;
AIN := (high - low)*temp2 / temp1 + low;

(* revision history
fixed an error with low value negative and high value 0.
hans
*)
END_FUNCTION

(* POU engineering/signal conditioning/Aout_16, ST *)
FUNCTION AOUT_16 : WORD
VAR_INPUT
	in : REAL;
END_VAR
VAR_INPUT CONSTANT
	Bits : BYTE;
	sign : BYTE := 255;
	low : REAL := 0;
	high : REAL := 10;
END_VAR
VAR
	temp : WORD;
	temp2 : WORD;
END_VAR

(*
version 1.0	4 aug 2006
programmer 	oscat
tested by		tobias

this module conditions an internal real value for a signal output D/A converter.
Aout_16 converts and internal real value to a word for an D/A converter or other output devices.
The input value is converted to a n-bit wide output and a sign bit is set separately as specified.
the outout min value is set for the specified min input value and the max output is set for the max input value.
an input higher or lower then the max or min value will set the respective max or min value or the output.


*) 
IF in < low THEN in := low;
ELSIF in > high THEN in := high;
END_IF;
temp := REAL_TO_WORD((in - low) / (high - low) * (EXPT(2,bits) -1));
IF sign_R(in) AND sign < 16 THEN
	temp := SHL(16#0001,sign) OR temp;
END_IF;
Aout_16 := temp;
END_FUNCTION

(* POU mathematical/sign_R, ST *)
FUNCTION sign_R : BOOL
VAR_INPUT
	in : REAL;
END_VAR
VAR
	X : DWORD;
END_VAR

(*
version 1.0	1 sep 2006
programmer 	hugo
tested by		tobias

this function return true if the real input is negative

*)
x := REAL_TO_DWORD(in);
sign_R := x.31;
END_FUNCTION

(* POU mathematical/array functions/array_avg, ST *)
FUNCTION array_avg : REAL
VAR_INPUT
	pt : POINTER TO ARRAY[0..32000] OF REAL;
	size : INT;
END_VAR
VAR
	i: INT;
	stop: INT;
END_VAR

(*
version 1.0	2 oct 2006
programmer 	hugo
tested by		tobias

this function will calculate the average of a given array.
the function needs to be called:	array_avg(adr("array"),sizeof("array"));
because this function works with pointers its very time efficient and it needs no extra memory.

*)
stop := (size -SIZEOF(pt)) / SIZEOF(pt);
array_avg := pt^[0];
FOR i := 1 TO stop DO
	array_avg := array_avg + pt^[i];
END_FOR;
array_avg := array_avg / (stop + 1);
END_FUNCTION

(* POU mathematical/array functions/array_max, ST *)
FUNCTION array_max : REAL
VAR_INPUT
	pt : POINTER TO ARRAY[0..32000] OF REAL;
	size : INT;
END_VAR
VAR
	i: INT;
	stop: INT;
END_VAR

(*
version 1.0	2 oct 2006
programmer 	hugo
tested by		tobias

this function will calculate the max value of a given array.
the function needs to be called:	array_max(adr("array"),sizeof("array"));
because this function works with pointers its very time efficient and it needs no extra memory.

*)
stop := (size -SIZEOF(pt)) / SIZEOF(pt);
array_max := pt^[0];
FOR i := 1 TO stop DO
	IF pt^[i] > array_max THEN array_max := pt^[i]; END_IF;
END_FOR;
END_FUNCTION

(* POU mathematical/array functions/array_min, ST *)
FUNCTION array_min : REAL
VAR_INPUT
	pt : POINTER TO ARRAY[0..32000] OF REAL;
	size : INT;
END_VAR
VAR
	i: INT;
	stop: INT;
END_VAR

(*
version 1.0	2 oct 2006
programmer 	hugo
tested by		tobias

this function will calculate the min value of a given array.
the function needs to be called:	array_min(adr("array"),sizeof("array"));
because this function works with pointers its very time efficient and it needs no extra memory.

*)
stop := (size - SIZEOF(pt)) / SIZEOF(pt);
array_min := pt^[0];
FOR i := 1 TO stop DO
	IF pt^[i] < array_min THEN array_min := pt^[i]; END_IF;
END_FOR;
END_FUNCTION

(* POU mathematical/array functions/array_spr, ST *)
FUNCTION array_spr : REAL
VAR_INPUT
	pt : POINTER TO ARRAY[0..32000] OF REAL;
	size : INT;
END_VAR
VAR
	i: INT;
	stop: INT;
	array_max : REAL;
	array_min : REAL;
END_VAR

(*
version 1.0	2 oct 2006
programmer 	hugo
tested by		tobias

this function will calculate the spread of a given array.
the function needs to be called:	array_spr(adr("array"),sizeof("array"));
for example: spread of [12,0,4,1,7] is 12 - 0 = 12.
because this function works with pointers its very time efficient and it needs no extra memory.

*)
stop := (size -SIZEOF(pt)) / SIZEOF(pt);
array_min := pt^[0];
array_max := pt^[0];
FOR i := 1 TO stop DO
	IF pt^[i] > array_max THEN array_max := pt^[i];
	ELSIF pt^[i] < array_min THEN array_min := pt^[i];
	END_IF;
END_FOR;
array_spr := array_max - array_min;
END_FUNCTION

(* POU mathematical/array functions/array_sum, ST *)
FUNCTION array_sum : REAL
VAR_INPUT
	pt : POINTER TO ARRAY[0..32000] OF REAL;
	size : INT;
END_VAR
VAR
	i: INT;
	stop: INT;
END_VAR


(*
version 1.0	2 oct 2006
programmer 	hugo
tested by		tobias

this function will calculate the sum of a given array.
the function needs to be called:	array_sum(adr("array"),sizeof("array"));
because this function works with pointers its very time efficient and it needs no extra memory.

*)
stop := (size -SIZEOF(pt)) / SIZEOF(pt);
array_sum := pt^[0];
FOR i := 1 TO stop DO
	array_sum := array_sum + pt^[i];
END_FOR;
END_FUNCTION

(* POU mathematical/array functions/array_trend, ST *)
FUNCTION array_trend : REAL
VAR_INPUT
	pt : POINTER TO ARRAY[0..32000] OF REAL;
	size : INT;
END_VAR
VAR
	i: INT;
	stop: INT;
	x: REAL;
	y : REAL;
END_VAR

(*
version 1.0	2 oct 2006
programmer 	hugo
tested by		tobias

this function will calculate the trend of a given array.
trend will calculate the avg of the first half of the array and then the avg of the second half, trend = avg2 - avg1.
for example:  [0,1,4,5,3,4,6,3] = 4 - 2.5 = 1.5
the function needs to be called:	array_trend(adr("array"),sizeof("array"));
because this function works with pointers its very time efficient and it needs no extra memory.

*)
stop := (size - SIZEOF(pt)) / SIZEOF(pt);
FOR i := 0 TO stop / 2 DO x := x + pt^[i]; END_FOR;
X := x / (TRUNC(stop / 2) + 1);
IF even(stop) THEN
	FOR i := stop / 2 TO stop DO y := y + pt^[i]; END_FOR;
	y := y / (stop / 2 + 1);
ELSE
	FOR i := TRUNC(stop / 2) + 1 TO stop DO y := y + pt^[i]; END_FOR;
	y := y / (TRUNC(stop / 2) + 1);
END_IF;
array_trend := y - x;
END_FUNCTION

(* POU Logic/generators/B_TRIG, ST *)
FUNCTION_BLOCK B_TRIG
VAR_INPUT
	CLK : BOOL;
END_VAR
VAR_OUTPUT
	Q : BOOL := 0;
END_VAR
VAR
	edge : BOOL := 0;
END_VAR

(*
version 1.0	4 aug 2006
programmer 	hugo
tested by		tobias

this block is similar to R_trig and F_trig but it generates a pulse on rising and falling edge.

executioin TIME on wago 750-841 = 5us
*)
Q := clk XOR edge;
edge := CLK;
END_FUNCTION_BLOCK

(* POU Logic/gate logic/Bit_of_Dword, ST *)
FUNCTION Bit_of_Dword : BOOL
VAR_INPUT
	in : DWORD;
	N : BYTE;
END_VAR
VAR
	temp: DWORD;
END_VAR

(*
version 1.0	4 aug 2006
programmer 	hugo
tested by		tobias

this function extracts a single bit from the nth position from right (right is lowest bit) *)
temp := SHR(in,n);
Bit_of_Dword := temp.0;
END_FUNCTION

(* POU Logic/gate logic/Bit_to_Byte, ST *)
FUNCTION Bit_to_Byte : BYTE
VAR_INPUT
	B0:BOOL;
	B1:BOOL;
	B2:BOOL;
	B3:BOOL;
	B4:BOOL;
	B5:BOOL;
	B6:BOOL;
	B7:BOOL;
END_VAR
VAR
	Bx : BYTE;
END_VAR

(*
version 1.0	4 aug 2006
programmer 	hugo
tested by		tobias

this function creates a byte from 8 individual bits

executioin TIME on wago 750-841 = 8 us
*)
BX.0 := B0;
BX.1 := B1;
BX.2 := B2;
BX.3 := B3;
BX.4 := B4;
BX.5 := B5;
BX.6 := B6;
BX.7 := B7;
bit_to_byte := BX;
END_FUNCTION

(* POU Logic/gate logic/Byte_to_Bit, ST *)
FUNCTION_BLOCK Byte_to_Bit
VAR_INPUT
	IN: BYTE;
END_VAR
VAR_OUTPUT
	B0: BOOL;
	B1: BOOL;
	B2: BOOL;
	B3: BOOL;
	B4: BOOL;
	B5: BOOL;
	B6: BOOL;
	B7: BOOL;
END_VAR
VAR
END_VAR

(*
version 1.0	4 aug 2006
programmer 	hugo
tested by		tobias

this Function Block extracts the 8 Bits from a byte

executioin TIME on wago 750-841 = 13us
*)
B0 := IN.0;
B1 := IN.1;
B2 := IN.2;
B3 := IN.3;
B4 := IN.4;
B5 := IN.5;
B6 := IN.6;
B7 := IN.7;
END_FUNCTION_BLOCK

(* POU engineering/conversion/C_to_F, ST *)
FUNCTION C_to_F : REAL
VAR_INPUT
	celsius : REAL;
END_VAR
VAR
END_VAR

(*
version 1.0	4 aug 2006
programmer 	hugo
tested by		tobias

this function converts celsius  to fahrenheit 

executioin TIME on wago 750-841 = 15us
*)
C_to_F := celsius * 1.8 + 32;
END_FUNCTION

(* POU Logic/gate logic/check_parity, ST *)
FUNCTION check_parity : BOOL
VAR_INPUT
	in : DWORD;
	p : BOOL;
END_VAR
VAR
	i: INT;
	cnt: INT := 0;
END_VAR

(*
version 1.0	1 oct 2006
programmer 	hugo
tested by		tobias

this function checks for an even partity for a dword and partity bit.

*)
FOR i := 0 TO 31 DO
	IF in.0 THEN cnt := cnt +1; END_IF;
	in := SHR(in,1);
END_FOR;
check_parity := even(cnt) XOR P;
END_FUNCTION

(* POU Logic/generators/CLK_1ms, ST *)
FUNCTION_BLOCK CLK_1ms
VAR_INPUT
END_VAR
VAR_OUTPUT
	Q : BOOL;
END_VAR
VAR
	CLK : BOOL;
	edge : BOOL := 0;
	stime: DWORD;
END_VAR

(*
clk_gen uses the internal sps time to generate one pulse every 1 ms
every pulse is only valid for one cycle so that a edge trigger is not necessary
clk_gen generates pulses depending on the accuracy of the system clock.

be careful, 1ms clocks will only work on very powerful sps cpu's
wago 750 - 841 will work with pulse width >= 10ms
*)
stime := TIME_TO_DWORD(TIME());
clk := stime.0;
Q := clk XOR edge;
edge := CLK;
END_FUNCTION_BLOCK

(* POU Logic/generators/CLK_2ms, ST *)
FUNCTION_BLOCK CLK_2ms
VAR_INPUT
END_VAR
VAR_OUTPUT
	Q : BOOL;
END_VAR
VAR
	CLK : BOOL;
	edge : BOOL := 0;
	stime: DWORD;
END_VAR

(*
clk_gen uses the internal sps time to generate one pulse every 2 ms
every pulse is only valid for one cycle so that a edge trigger is not necessary
clk_gen generates pulses depending on the accuracy of the system clock.

be careful, 1ms clocks will only work on very powerful sps cpu's
wago 750 - 841 will work with pulse width >= 10ms
*)
stime := TIME_TO_DWORD(TIME());
clk := stime.1;
Q := clk XOR edge;
edge := CLK;
END_FUNCTION_BLOCK

(* POU Logic/generators/CLK_4ms, ST *)
FUNCTION_BLOCK CLK_4ms
VAR_INPUT
END_VAR
VAR_OUTPUT
	Q : BOOL;
END_VAR
VAR
	CLK : BOOL;
	edge : BOOL := 0;
	stime: DWORD;
END_VAR

(*
clk_gen uses the internal sps time to generate one pulse every 4 ms
every pulse is only valid for one cycle so that a edge trigger is not necessary
clk_gen generates pulses depending on the accuracy of the system clock.

be careful, 1ms clocks will only work on very powerful sps cpu's
wago 750 - 841 will work with pulse width >= 10ms
*)
stime := TIME_TO_DWORD(TIME());
clk := stime.2;
Q := clk XOR edge;
edge := CLK;
END_FUNCTION_BLOCK

(* POU Logic/generators/CLK_8ms, ST *)
FUNCTION_BLOCK CLK_8ms
VAR_INPUT
END_VAR
VAR_OUTPUT
	Q : BOOL;
END_VAR
VAR
	CLK : BOOL;
	edge : BOOL := 0;
	stime: DWORD;
END_VAR

(*
clk_gen uses the internal sps time to generate one pulse every 8 ms
every pulse is only valid for one cycle so that a edge trigger is not necessary
clk_gen generates pulses depending on the accuracy of the system clock.

be careful, 1ms clocks will only work on very powerful sps cpu's
wago 750 - 841 will work with pulse width >= 10ms
*)
stime := TIME_TO_DWORD(TIME());
clk := stime.3;
Q := clk XOR edge;
edge := CLK;
END_FUNCTION_BLOCK

(* POU Logic/generators/clk_div, ST *)
FUNCTION_BLOCK clk_div
VAR_INPUT
	clk : BOOL;
	rst: BOOL;
END_VAR
VAR_OUTPUT
	Q0 : BOOL := 0;
	Q1 : BOOL := 0;
	Q2 : BOOL := 0;
	Q3 : BOOL := 0;
	Q4 : BOOL := 0;
	Q5 : BOOL := 0;
	Q6 : BOOL := 0;
	Q7 : BOOL := 0;
END_VAR
VAR
	cnt: BYTE := 0;
END_VAR

(*
version 1.0	4 aug 2006
programmer 	hugo
tested by		tobias

this is a clock divider
each output divides the signal by 2
Q0 = clk / 2 , Q1 = Q0 / 2 and so on.
the outputs have a 50% duty cycle each.


*)
IF clk AND NOT rst THEN
	cnt:= cnt +1;
	Q0 := cnt.0;
	Q1 := cnt.1;
	Q2 := cnt.2;
	Q3 := cnt.3;
	Q4 := cnt.4;
	Q5 := cnt.5;
	Q6 := cnt.6;
	Q7 := cnt.7;
END_IF;
IF rst THEN
	cnt:= 0;
	Q0 := 0;
	Q1 := 0;
	Q2 := 0;
	Q3 := 0;
	Q4 := 0;
	Q5 := 0;
	Q6 := 0;
	Q7 := 0;
END_IF;
END_FUNCTION_BLOCK

(* POU Logic/generators/CLK_Prg, ST *)
FUNCTION_BLOCK CLK_Prg
VAR_INPUT
	PT : TIME := t#10ms;
END_VAR
VAR_OUTPUT
	Q : BOOL := 0;
END_VAR
VAR
	pti : TIME := t#0ms;
	next_pulse: TIME := T#0s;
	run: BOOL := FALSE;
	overflow: BOOL := FALSE;
END_VAR

(*
version 1.0	4 aug 2006
programmer 	hugo
tested by		tobias

clk_prg uses the internal sps time to generate a clock with programmable period time.
the period time is defined for 10ms .. 65s
if the period time is set to less then 10ms the min clock perid is 10ms.
the first cycle after start is a clk pulse and then depending on the programmed period time a delay.
every pulse is only valid for one cycle so that a edge trigger is not necessary
clk_prg depending on the accuracy of the system clock.

*)
IF NOT run THEN
	next_pulse := TIME();
	run := TRUE;
	IF pt < T#10ms THEN PTI := T#10ms; ELSE pti := pt; END_IF;
END_IF;
IF TIME() >= next_pulse AND NOT overflow THEN
	Q := TRUE;
	IF next_pulse + pti < next_pulse THEN
		overflow := TRUE;
	END_IF;
	next_pulse := next_pulse + pti;
ELSE
	Q := FALSE;
	IF TIME() <= next_pulse THEN overflow := FALSE; END_IF;
END_IF;
END_FUNCTION_BLOCK

(* POU Logic/generators/CLK_Pulse, ST *)
FUNCTION_BLOCK CLK_Pulse
VAR_INPUT
	PT : TIME := t#10ms;
	N : INT := 0;
	rst : BOOL := 0;
END_VAR
VAR_OUTPUT
	Q : BOOL := 0;
	cnt : INT := 0;
	run : BOOL := 0;
END_VAR
VAR
	pti : TIME := t#0ms;
	next_pulse: TIME := T#0s;
	overflow: BOOL := FALSE;
END_VAR

(*
version 1.0	4 aug 2006
programmer 	hugo
tested by		tobias

clk_pulse uses the internal sps time to generate a clock with programmable period time.
the period time is defined for 10ms .. 65s.
pulse generation is continuous if N = 0 and for n pulses otherwise.
if the period time is set to less then 10ms the min clock perid is 10ms.
the first cycle after start is a clk pulse and then depending on the programmed period time a delay.
every pulse is only valid for one cycle so that a edge trigger is not necessary
clk_prg depending on the accuracy of the system clock.

*)
IF rst THEN
	run := FALSE;
	pti := t#0ms;
	next_pulse := t#0ms;
	overflow := FALSE;
	Q := FALSE;
	cnt := 0;
ELSIF cnt <= N OR N = 0 THEN
	IF NOT run THEN
		next_pulse := TIME();
		run := TRUE;
		IF pt < T#10ms THEN PTI := T#10ms; ELSE pti := pt; END_IF;
	END_IF;
	IF TIME() >= next_pulse AND NOT overflow AND (cnt < N OR N = 0) THEN
		Q := TRUE;
		cnt := cnt + 1;
		IF next_pulse + pti < next_pulse THEN
			overflow := TRUE;
		END_IF;
		next_pulse := next_pulse + pti;
	ELSE
		Q := FALSE;
		IF cnt = N THEN run := FALSE; END_IF
		IF TIME() <= next_pulse THEN overflow := FALSE; END_IF;
	END_IF;
END_IF
END_FUNCTION_BLOCK

(* POU Time&Date/day_of_month, ST *)
FUNCTION day_of_month : INT
VAR_INPUT
	idate : DATE;
END_VAR
VAR
	yd: INT;
	day_in_year: DWORD;
	day_in_year_begin: DWORD;
	yr: INT;
END_VAR

(*
version 1.0	4 aug 2006
programmer 	hugo
tested by		tobias

returns the day OF month from any DATE
execution TIME with wago 750-841 = 65 us
*)
yr := DWORD_TO_INT((DATE_TO_DWORD(idate)/864+71954300)/36525);
yd := DWORD_TO_INT(DATE_TO_DWORD(idate)/86400 - TRUNC((yr-1)*365.25) + 719178);
IF yr MOD 4 = 0 THEN
	CASE yd OF
		1..31 	:	day_of_month := yd;
		32..60	:	day_of_month := yd - 31;
		61..91	:	day_of_month := yd - 60;
		92..121 :	day_of_month := yd - 91;
		122..152:	day_of_month := yd - 121;
		153..182:	day_of_month := yd - 152;
		183..213:	day_of_month := yd - 182;
		214..244:	day_of_month := yd - 213;
		245..274:	day_of_month := yd - 244;
		275..305:	day_of_month := yd - 274;
		306..335:	day_of_month := yd - 305;
		336..366:	day_of_month := yd - 335;
	END_CASE;
	ELSE
	CASE yd OF
		1..31 	:	day_of_month := yd;
		32..59	:	day_of_month := yd - 31;
		60..90	:	day_of_month := yd - 59;
		91..120 :	day_of_month := yd - 90;
		121..151:	day_of_month := yd - 120;
		152..181:	day_of_month := yd - 151;
		182..212:	day_of_month := yd - 181;
		213..243:	day_of_month := yd - 212;
		244..273:	day_of_month := yd - 243;
		274..304:	day_of_month := yd - 273;
		305..334:	day_of_month := yd - 304;
		335..365:	day_of_month := yd - 334;
	END_CASE;
	END_IF;




(*
this function is simple but took too long with 133 us
the problem is date_to_string is far too slow
day_of_month := STRING_TO_INT(RIGHT(DATE_TO_STRING(idate),2));
*)
END_FUNCTION

(* POU Time&Date/day_of_year, ST *)
FUNCTION day_of_year : INT
VAR_INPUT
	idate : DATE;
END_VAR
VAR
END_VAR

(*
version 1.0	4 aug 2006
programmer 	hugo
tested by		tobias

calculates the day of the year 
execution time for wago 750-841 = 44 us  
*)
day_of_year := DWORD_TO_INT(DATE_TO_DWORD(idate)/86400 + 719178 - TRUNC((year(idate)-1)*365.25));
END_FUNCTION

(* POU Time&Date/year, ST *)
FUNCTION year : INT
VAR_INPUT
	idate : DATE;
END_VAR
VAR
END_VAR

(*
version 1.0	4 aug 2006
programmer 	hugo
tested by		tobias

returs the year of a date  
the function works for dates from 1970 - 2099 
execution time on wago 750-841 = 20us   
*)
year := DWORD_TO_INT((DATE_TO_DWORD(idate)/864+71954300)/36525);
END_FUNCTION

(* POU Time&Date/day_to_time, ST *)
FUNCTION day_to_time : TIME
VAR_INPUT
	input : REAL;
END_VAR
VAR
END_VAR

(*
version 1.0	4 aug 2006
programmer 	hugo
tested by		tobias

converts an amount of days in real to time 
execution time on wago 750-841 =  17 us 
*)
day_to_time := DWORD_TO_TIME(REAL_TO_DWORD(input * 86400000));
END_FUNCTION

(* POU Time&Date/DCF77, ST *)
FUNCTION_BLOCK DCF77
VAR_INPUT
	rec : BOOL;
END_VAR
VAR_INPUT CONSTANT
	sync_timeout : TIME := t#2m;
	time_offset : TIME := t#1h;
	dst_en : BOOL := TRUE;
END_VAR
VAR_OUTPUT
	TP : BOOL;
	DST : BOOL;
	weekday : INT;
	error: BOOL := TRUE;
	RTC : DT;
	RTC1 : DT;
	msec : INT;
	sync : BOOL;
END_VAR
VAR
	MEZ : DT;
	UTC : DT;
	state : INT;
	edge: BOOL;
	tx : TIME;
	ty: TIME;
	last : TIME;
	bits : ARRAY[0..58] OF BOOL;
	cnt : INT;
	i : INT;
	old_time : DT;
	minute : INT;
	hour : INT;
	day : INT;
	month : INT;
	year : INT;
	last_sync: TIME;
END_VAR


(*
version 1.0	2 oct 2006
programmer 	hugo
tested by		tobias

this is a decoder for a DCF77 signal.
the decoder decodes the DCF77 signal and checks for a valid Date_Time.
since the dcf77 signal is only secured with a simple parity the decoder waits for two consecutive valid transmissions before it sets the output signals.
given a valid reception by the receiver the decoder can take up to 3 minutes to start its clocks the first time.
after a valid signal is detected the error output goes low and dignals a valid dcf signal from the receiver.
a tp is only valid for one program cycle to allow for external rtc setting.
after a valid signal is detected two independent internal clocks are started (RTC and RTC1), the seconds  of these clocks are generated by software since the dcf signal is only valid for minutes.
rtc is always utc ( world time) and rtc1 can be set to any time zone by setting the time_zone_offset and enabling dst for automatic summertime.
a sync output signals the the rtc and rtc1 are in sync with the dcf77 signal, if the dcf77 signal is lost for more then the sync time the sync output goes low
but the rtc and rtc1 outputs keep running based on software timing until a valid dcf77 signal is received again and triggers the clock.
in addition a millisecond output gives further resolutionof the clocks.
a dst output shows if daylight saving time is enables and the weekday output shows which day of week currently is ( 1= monday ... 7= sunday).


*)
(* if tp was set it should only be active for 1 cycle *)
TP := FALSE;
IF rec XOR edge THEN
	tx := TIME() - last;
	edge := rec;
	IF NOT rec AND tx > t#1700ms AND tx < t#2000ms THEN
		(* start condition reached *)
		state := 0;
		tp := NOT error;
	ELSIF NOT rec AND tx > t#700ms AND tx < t#1000ms THEN
		(* second switch detected *)
		IF state < 58 THEN state := state +1; ELSE state := 0; END_IF;
	ELSIF rec AND tx  < t#120ms THEN
		(* bit 0 detected  *)
		bits[state] := 0;
	ELSIF rec AND tx > t#120ms AND tx < t#250ms THEN
		(* bit 1 detected *)
		bits[state] := 1;
	ELSE
		(* error condition received signal is not valid *)
		error := TRUE;
		state := 0;
	END_IF;
	last := last + tx;
	IF rec AND state = 58 THEN
		error := FALSE;
		(* decode the bits and check for possible errors *)
		IF bits[0] OR NOT (bits[17] XOR bits[18]) OR NOT bits[20] THEN error := TRUE; END_IF;
		(* decode minute *)
		minute := 0;
		minute.0 := bits[21];
		minute.1 := bits[22];
		minute.2 := bits[23];
		minute.3 := bits[24];
		IF bits[25] THEN minute := minute + 10; END_IF;
		IF bits[26] THEN minute := minute +20; END_IF;
		IF bits[27] THEN minute := minute +40; END_IF;
		IF minute > 59 OR (bits[21] XOR bits[22] XOR bits[23] XOR bits[24] XOR bits[25] XOR bits[26] XOR bits[27] XOR bits[28]) THEN error := TRUE; END_IF;

		(* decode hour *)
		hour := 0;
		hour.0 := bits[29];
		hour.1 := bits[30];
		hour.2 := bits[31];
		hour.3 := bits[32];
		IF bits[33] THEN hour := hour + 10; END_IF;
		IF bits[34] THEN hour := hour +20; END_IF;
		IF hour > 23 OR (bits[29] XOR bits[30] XOR bits[31] XOR bits[32] XOR bits[33] XOR bits[34] XOR bits[35]) THEN error := TRUE; END_IF;

		(* decode day of month *)
		day := 0;
		day.0 := bits[36];
		day.1 := bits[37];
		day.2 := bits[38];
		day.3 := bits[39];
		IF bits[40] THEN day := day + 10; END_IF;
		IF bits[41] THEN day := day + 20; END_IF;
		IF day > 31 THEN error := TRUE; END_IF;

		(* decode day of week *)
		weekday := 0;
		weekday.0 := bits[42];
		weekday.1 := bits[43];
		weekday.2 := bits[44];
		IF weekday > 7 OR weekday < 1 THEN error := TRUE; END_IF;

		(* decode month *)
		month := 0;
		month.0 := bits[45];
		month.1 := bits[46];
		month.2 := bits[47];
		month.3 := bits[48];
		IF bits[49] THEN month := month +10; END_IF;
		IF month > 12 THEN error := TRUE; END_IF;

		(* decode year *)
		year := 0;
		year.0 := bits[50];
		year.1 := bits[51];
		year.2 := bits[52];
		year.3 := bits[53];
		IF bits[54] THEN year := year + 10; END_IF;
		IF bits[55] THEN year := year + 20; END_IF;
		IF bits[56] THEN year := year + 40; END_IF;
		IF bits[57] THEN year := year + 80; END_IF;

		(* check parity for bits 36 to 58 *)
		cnt := 0;
		FOR i := 36 TO 58 DO IF bits[i] THEN cnt := cnt + 1; END_IF; END_FOR;
		IF NOT even(cnt) THEN error := TRUE; END_IF;

		(* time must be valid for two cycles to clear error flag *)
		IF NOT error THEN
			(* set outputs *)
			old_time := mez;
			IF year >= 70 THEN year := year + 1900; ELSE year := year + 2000; END_IF;
			mez := set_DT(year,month,day,hour,minute,0);
			DST := bits[17];
			IF DST THEN UTC := mez - t#2h; ELSE utc := mez - t#1h; END_IF;
			(* set trigger signal only if the receiver has received 2 successive minutes *)
			IF mez <> old_time + t#1m THEN error := TRUE ; END_IF;
		END_IF;
	END_IF;
END_IF;

(* this portion implements a free running clock which is triggered by the dcf77 signal *)
IF tp THEN
	rtc := utc;
	IF DST AND dst_en THEN rtc1 := rtc + time_offset + t#1h; ELSE rtc1 := rtc + time_offset; END_IF;
	sync := TRUE;
	last_sync := last;
	ty := last;
ELSIF rtc > DWORD_TO_DT(0) AND TIME() - ty >= t#1s THEN
	rtc := rtc + t#1s;
	rtc1 := rtc1 + t#1s;
	ty := ty + t#1s;
	sync := ty - last_sync < sync_timeout AND last_sync > DWORD_TO_TIME(0);
END_IF;
msec := TIME_TO_INT(TIME() - ty);



(* decode information
bits		content
0			Bitwert immer 0
1 bis 14	reserviert für Betriebsinformationen (nicht für DCF77-Nutzer bestimmt)
15			Rufbit für Alarmierung der PTB-Mitarbeiter
			(bis Mai 2003: Bitwert = 0 falls normale Antenne in Verwendung; 1 = Backupantenne)
16			Bitwert = 1 falls ein Wechsel von MEZ nach MESZ oder umgekehrt bevorsteht; Dauer der Anzeige: 1 Stunde
17 + 18	gültige Zeit = MEZ, falls Bit 17=0 und Bit 18=1
			gültige Zeit = MESZ, falls Bit 17=1 und Bit 18=0
19			Bitwert = 1 falls innerhalb den nächsten 59 Minuten eine Schaltsekunde angeordnet ist. Beim Einfügen einer Schaltsekunde wird anstelle der 59. die 60. Sekundenmarke weggelassen und in der 58. erfolgt ausnahmsweise ein Trägerabfall.
20			Startbit für Zeitinformation (immer 1)
21 - 27		1, 2, 4, 8, 10, 20, 40 Minuten (bitweise Addition)
28			Prüfbit (gerade Parität) für die Bits 21-27
29 - 34		1, 2, 4, 8, 10, 20 Stunden (bitweise Addition)
35			Prüfbit (gerade Parität) für die Bits 29-34
36 - 41		Tagesnummer im aktuellen Monat: 1, 2, 4, 8, 10, 20 (bitweise Addition)
42 - 44		Tagesnummer in der aktuellen Woche: 1, 2, 4 (bitweise Addition)
45 - 49		Monatsnummer: 1, 2, 4, 8, 10 (bitweise Addition)
50 - 57		Jahr (zweistellig): 1, 2, 4, 8, 10, 20, 40, 80 (bitweise Addition)
58			Prüfbit (gerade Parität) füR die Bits 36-57

*)
END_FUNCTION_BLOCK

(* POU Time&Date/DST, ST *)
FUNCTION DST : BOOL
VAR_INPUT
	utc : DT;
	time_zone_offset : TIME;
END_VAR
VAR
	yr : INT;
	yr4 : DWORD;
	ltc: DWORD;
	idate : DWORD;
END_VAR

(*
version 1.0	4 aug 2006
programmer 	hugo
tested by		tobias

 this functions returns TRUE IF dst TIME is active 
 the FUNCTION calculates automaticall FOR any year betweek 1970 AND 2099 
wheather daylight savings is on OR off 
the summertime calculation is done according to european standards.
dst will become TRUE AT 02:00 in the morning FOR the respective days 
AND it will become FALSE after daylight savings TIME is switched back end OF october automatically 
(execution TIME on wago 750-841 =  110us   
*)
yr := year(DT_TO_DATE(utc));
ltc := DT_TO_DWORD(utc+time_zone_offset);
idate := DT_TO_DWORD(set_DT(yr,3,31,2,0,0));
yr4 := 5*yr/4;
IF idate - ((yr4+4) MOD 7)*86400 <= ltc AND idate + (214 - (yr4+1) MOD 7)*86400 > ltc THEN DST := TRUE; ELSE DST := FALSE; END_IF;


(*

Equation used TO calculate the beginning OF European Summer TIME:
Sunday (31 - (5*y/4 + 4) mod 7) March at 01.00 UTC
(valid through 2099, courtesy of Robert H. van Gent, EC).

European Summer Time ends (clocks go back) at 01.00 UTC on

    * 29 October 2006
    * 28 October 2007
    * 26 October 2008

Equation used to calculate the end of European Summer Time:
Sunday (31 - (5*y/4 + 1) mod 7) October at 01.00 UTC
(validity AND credits as above).

*)
END_FUNCTION

(* POU Time&Date/set_DT, ST *)
FUNCTION set_DT : DT
VAR_INPUT
	year : INT;
	month : INT;
	day : INT;
	hour : INT;
	minute : INT;
	second : INT;
END_VAR
VAR
	count : DWORD;
	leap : BOOL;
END_VAR

(*
version 1.0	4 aug 2006
programmer 	hugo
tested by		tobias


creates a date output from year, month and day of month
year must be in the form of 4 digits ie 2006 or 1977.
execution time on wago 750-841 = 45 us   
*)
IF year MOD 4 = 0 THEN leap := TRUE; ELSE leap := FALSE; END_IF;
count := TRUNC((year-1)*365.25-719178+day);
CASE month OF
2:	count := count + 31;
3:	IF leap THEN count := count + 60; ELSE count := count + 59; END_IF;
4:	IF leap THEN count := count + 91; ELSE count := count + 90; END_IF;
5:	IF leap THEN count := count + 121; ELSE count := count + 120; END_IF;
6:	IF leap THEN count := count + 152; ELSE count := count + 151; END_IF;
7:	IF leap THEN count := count + 182; ELSE count := count + 181; END_IF;
8:	IF leap THEN count := count + 213; ELSE count := count + 212; END_IF;
9:	IF leap THEN count := count + 244; ELSE count := count + 243; END_IF;
10:	IF leap THEN count := count + 274; ELSE count := count + 273; END_IF;
11:	IF leap THEN count := count + 305; ELSE count := count + 304; END_IF;
12:	IF leap THEN count := count + 335; ELSE count := count + 334; END_IF;
END_CASE;
set_DT := DWORD_TO_DT(count * 86400 + second + minute * 60 + hour * 3600);
END_FUNCTION

(* POU Time&Date/month, ST *)
FUNCTION month : INT
VAR_INPUT
	idate : DATE;
END_VAR
VAR
END_VAR

(*
version 1.0	4 aug 2006
programmer 	hugo
tested by		tobias

returns the month of a date  
execution time on wago 750-841 = 145us
*)
month := STRING_TO_INT(MID(DATE_TO_STRING(idate),2,8));
END_FUNCTION

(* POU Time&Date/hour, ST *)
FUNCTION hour : INT
VAR_INPUT
	itod : TOD;
END_VAR
VAR
END_VAR

(*
version 1.0	4 aug 2006
programmer 	hugo
tested by		tobias

extracts the hour of a Time_of_day 
execution time for wago 750-841 = 10 us  
*)
hour := DWORD_TO_INT(TOD_TO_DWORD(itod)/3600000);




(* change history

2.10.2006 changes name of input to itod

*)
END_FUNCTION

(* POU Time&Date/minute, ST *)
FUNCTION minute : INT
VAR_INPUT
	itod : TOD;
END_VAR
VAR
END_VAR

(*
version 1.1	2 oct 2006
programmer 	hugo
tested by		tobias

extracts the minutes out of TOD truncating the ceconds 
execution time on wago 750-841  = 18us

*)  
minute := DWORD_TO_INT(TOD_TO_DWORD(itod)/60000 - TOD_TO_DWORD(itod)/3600000 * 60);


(* change history

2.10.2006 changes name of input to itod

*)
END_FUNCTION

(* POU Time&Date/second, ST *)
FUNCTION second : REAL
VAR_INPUT
	itod : TOD;
END_VAR
VAR
END_VAR

(*
version 1.1	2 oct 2006
programmer 	hugo
tested by		tobias

returns the seconds and milliseconds as real of TOD   
execution time on wago 750-841 = 20 us 
*)
second := DWORD_TO_REAL(TOD_TO_DWORD(itod) - TOD_TO_DWORD(itod)/60000 * 60000)/1000;



(* change history

2.10.2006 changes name of input to itod

*)
END_FUNCTION

(* POU Time&Date/weekday, ST *)
FUNCTION weekday : INT
VAR_INPUT
	idate : DATE;
END_VAR
VAR
END_VAR

(*
version 1.1	21 aug 2006
programmer 	hugo
tested by		tobias

calculates the weekday of a week   
monday = 1 ..... sunday = 7  
execution time on wago 750-841 = 22 us  
*)
weekday := DWORD_TO_INT((DATE_TO_DWORD(idate)/86400+3) MOD 7)+1;

(* corrected a miscalculation formula is now correct *)
END_FUNCTION

(* POU Logic/gate logic/DEC_2, CFC *)
FUNCTION_BLOCK DEC_2
VAR_INPUT
	D: BOOL;
	A: BOOL;
END_VAR
VAR_OUTPUT
	Q0: BOOL;
	Q1: BOOL;
END_VAR
VAR
END_VAR

(*
version 1.0	4 aug 2006
programmer 	hugo
tested by		tobias

a bit input will be decoded to the two outputs Q0 or Q1
dependent on the value of A
A=0 decodes to Q0 and A=1 decodes to Q1

executioin TIME on wago 750-841 = 5us
*)
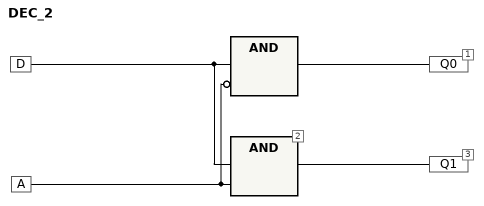
_CFC_ (* Continuous Function Chart, elements in execution order *)
#0 AND(D, NOT A)
#1 Q0 <= #0
#2 AND(D, A)
#3 Q1 <= #2
_END_CFC_
(* the same logic as Structured Text *)
Q0 := D AND NOT A;
Q1 := D AND A;
END_FUNCTION_BLOCK

(* POU Logic/gate logic/DEC_4, CFC *)
FUNCTION_BLOCK DEC_4
VAR_INPUT
	D: BOOL;
	A0: BOOL;
	A1: BOOL;
END_VAR
VAR_OUTPUT
	Q0: BOOL;
	Q1: BOOL;
	Q2: BOOL;
	Q3: BOOL;
END_VAR
VAR
END_VAR

(*
version 1.0	4 aug 2006
programmer 	hugo
tested by		tobias

a bit input will be decoded to one of the 4 outputs
dependent on the Adress on A0 and A1

executioin TIME on wago 750-841 = 9us
*)
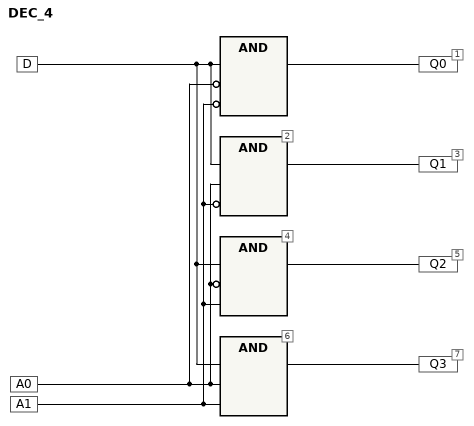
_CFC_ (* Continuous Function Chart, elements in execution order *)
#0 AND(D, NOT A0, NOT A1)
#1 Q0 <= #0
#2 AND(D, A0, NOT A1)
#3 Q1 <= #2
#4 AND(D, NOT A0, A1)
#5 Q2 <= #4
#6 AND(D, A0, A1)
#7 Q3 <= #6
_END_CFC_
(* the same logic as Structured Text *)
Q0 := D AND NOT A0 AND NOT A1;
Q1 := D AND A0 AND NOT A1;
Q2 := D AND NOT A0 AND A1;
Q3 := D AND A0 AND A1;
END_FUNCTION_BLOCK

(* POU Logic/gate logic/DEC_8, CFC *)
FUNCTION_BLOCK DEC_8
VAR_INPUT
	D: BOOL;
	A0: BOOL;
	A1: BOOL;
	A2: BOOL;
END_VAR
VAR_OUTPUT
	Q0: BOOL;
	Q1: BOOL;
	Q2: BOOL;
	Q3: BOOL;
	Q4: BOOL;
	Q5: BOOL;
	Q6: BOOL;
	Q7: BOOL;
END_VAR
VAR
END_VAR

(*
version 1.0	4 aug 2006
programmer 	hugo
tested by		tobias

a bit input will be decoded to one of the 8 outputs
dependent on the Adress on A0, A1 and A2

executioin TIME on wago 750-841 = 17us
*)
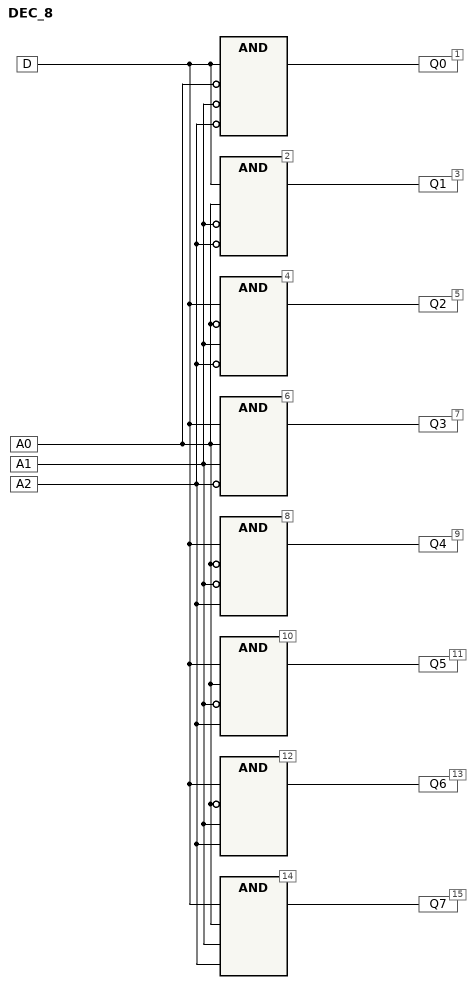
_CFC_ (* Continuous Function Chart, elements in execution order *)
#0 AND(D, NOT A0, NOT A1, NOT A2)
#1 Q0 <= #0
#2 AND(D, A0, NOT A1, NOT A2)
#3 Q1 <= #2
#4 AND(D, NOT A0, A1, NOT A2)
#5 Q2 <= #4
#6 AND(D, A0, A1, NOT A2)
#7 Q3 <= #6
#8 AND(D, NOT A0, NOT A1, A2)
#9 Q4 <= #8
#10 AND(D, A0, NOT A1, A2)
#11 Q5 <= #10
#12 AND(D, NOT A0, A1, A2)
#13 Q6 <= #12
#14 AND(D, A0, A1, A2)
#15 Q7 <= #14
_END_CFC_
(* the same logic as Structured Text *)
Q0 := D AND NOT A0 AND NOT A1 AND NOT A2;
Q1 := D AND A0 AND NOT A1 AND NOT A2;
Q2 := D AND NOT A0 AND A1 AND NOT A2;
Q3 := D AND A0 AND A1 AND NOT A2;
Q4 := D AND NOT A0 AND NOT A1 AND A2;
Q5 := D AND A0 AND NOT A1 AND A2;
Q6 := D AND NOT A0 AND A1 AND A2;
Q7 := D AND A0 AND A1 AND A2;
END_FUNCTION_BLOCK

(* POU mathematical/deg, ST *)
FUNCTION deg : REAL
VAR_INPUT
	rad : REAL;
END_VAR
VAR
END_VAR
VAR
END_VAR

(*
version 1.0	4 aug 2006
programmer 	hugo
tested by		tobias

this function converts degrees into Radiant
execution time on wago 750 - 841 =  10  us
*)
deg := 57.29577951308232 * Rad;
END_FUNCTION

(* POU mathematical/Rad, ST *)
FUNCTION Rad : REAL
VAR_INPUT
	deg : REAL;
END_VAR
VAR
END_VAR

(*
version 1.0	4 aug 2006
programmer 	hugo
tested by		tobias

this function converts Radiant to degrees
execution time on wago 750 - 841 =  10  us
*)
Rad := 0.0174532925199433 * deg;
END_FUNCTION

(* POU engineering/signal conditioning/delay, ST *)
FUNCTION_BLOCK delay
VAR_INPUT
	in : REAL;
	N : INT;
	rst : BOOL;
END_VAR
VAR_OUTPUT
	out : REAL;
END_VAR
VAR
	buf : ARRAY[0..31] OF REAL;
	i : INT;
END_VAR

(*
version 1.1	1. oct. 2006
programmer 	hugo
tested by		tobias

this function block delays input values by each programm cycle
after N+1 cycles the in value has shifted to the out.
N can be any alue from 0 .. 32
if n = 0 the input will be present on the output without a delay.
f N > 32 then the output will be delayed by 32 cycles.
any high on rst will clear the buffer.

*)
IF N > SIZEOF(buf) / SIZEOF(in) THEN N:= 32; END_IF;
IF rst THEN
	FOR i := 0 TO 31 DO buf[i] := 0; END_FOR;
	out := 0;
ELSIF N < 1 THEN out := in;
ELSE
	IF i >= N THEN i := 0; END_IF;
	out := buf[i];
	buf[i] := in;
	i := i + 1;
END_IF;
END_FUNCTION_BLOCK

(* POU engineering/signal conditioning/delay_4, ST *)
FUNCTION_BLOCK delay_4
VAR_INPUT
	in : REAL;
END_VAR
VAR_OUTPUT
	out1 : REAL;
	out2 : REAL;
	out3 : REAL;
	out4 : REAL;
END_VAR
VAR
END_VAR

(*
version 1.0	1 sep 2006
programmer 	hugo
tested by		tobias

this function block delays input values by each programm cycle
after 4 cycles the in value has shifted to the out 4 and will be discarded after the next cycle
the blocks can be cascaded.

*)
out4 := out3;
out3 := out2;
out2 := out1;
out1 := in;
END_FUNCTION_BLOCK

(* POU Building/HLK/dew_temp, ST *)
FUNCTION dew_temp : REAL
VAR_INPUT
	RH : REAL;
	T : REAL;
END_VAR
VAR
	a : REAL := 7.5;
	b : REAL := 237.3;
	SDD : REAL;
	DD : REAL;
	V : REAL;
END_VAR

(*
version 1.0	2 oct 2006
programmer 	hugo
tested by		tobias

this function calculates the deew point for air given the temperature and relative humidity.
dew_temp(60,25) = 16.7 °C.
which means the dew point for air with 25° and 60% RH is at 16.7 °C.


*)
SDD := 6.1078*EXPT(10,(a*T)/(b+T));
DD := RH/100 * SDD;
V := LOG(DD/6.1078);
dew_temp := b*V/(a-v);

(*
Bezeichnungen:
r = relative Luftfeuchte
T = Temperatur in °C
TK = Temperatur in Kelvin (TK = T + 273.15)
TD = Taupunkttemperatur in °C
DD = Dampfdruck in hPa
SDD = Sättigungsdampfdruck in hPa

Parameter:
a = 7.5, b = 237.3 für T >= 0
a = 7.6, b = 240.7 für T < 0 über Wasser (Taupunkt)
a = 9.5, b = 265.5 für T < 0 über Eis (Frostpunkt)

R* = 8314.3 J/(kmol*K) (universelle Gaskonstante)
mw = 18.016 kg (Molekulargewicht des Wasserdampfes)
AF = absolute Feuchte in g Wasserdampf pro m3 Luft

Formeln:

   1. SDD(T) = 6.1078 * 10^((a*T)/(b+T))
   2. DD(r,T) = r/100 * SDD(T)
   3. r(T,TD) = 100 * SDD(TD) / SDD(T)
   4. TD(r,T) = b*v/(a-v) mit v(r,T) = log10(DD(r,T)/6.1078)
   5. AF(r,TK) = 10^5 * mw/R* * DD(r,T)/TK; AF(TD,TK) = 10^5 * mw/R* * SDD(TD)/TK 

*)
END_FUNCTION

(* POU Building/dimm_i, ST *)
FUNCTION_BLOCK dimm_i
VAR_INPUT
	set : BOOL;
	in : BOOL;
	rst : BOOL;
END_VAR
VAR_INPUT CONSTANT
	T_debounce : TIME := T#10ms;
	T_reconfig : TIME := T#10s;
	T_on_max : TIME := T#0h;
	T_dimm_start : TIME := T#1s;
	T_dimm: TIME := T#3s;
END_VAR
VAR_OUTPUT
	Q : BOOL := 0;
	out : BYTE := 0;
END_VAR
VAR
	tx : TIME := T#0s;
	last_edge : BOOL;
	state : BYTE := 0;
	edge : BOOL := 0;
	r_edge : BOOL := 0;
	T_on : TIME;
	dimm_up: BOOL;
	ramp : rmp_B;
	last_step : TIME;
END_VAR

(*
version 1.0	4 aug 2006
programmer 	hugo
tested by		tobias

this is an intelligent dimmer interface with an autoset feature for "in" it will automatically detect the type of switch:
low active pulses or high high active pulses are allowd for in.
a configurable debounce timer will debounce input signals
if t_on_max is set to anything other then 0 the output will be turned off after the max on time is reached.
the times for debounce, dimming ramp, wait time before dimming and max on time are all programmable.

the dimmer has outputs Q for on and off and also out with the analog dimm value.

*)
IF rst THEN
	state := 0;
	Q := 0;
	dimm_up := TRUE;
ELSIF set THEN
	state := 0;
	Q := TRUE;
	out := 255;
	dimm_up := FALSE;
	T_on := TIME();
ELSE
	CASE state OF
	(* state 0 wait for activity *)
	0 :	IF (r_edge AND in AND NOT edge) OR (NOT r_edge AND NOT in AND edge) THEN
			state := 1;
			tx := TIME();
			last_edge := in;
		END_IF

	(* state 1 debouncing *)
	1:	IF TIME() - T_debounce >= tx THEN
			state := 2;
			tx := TIME();
		END_IF;

	(* state 2 wait for second edge to toggle output *)
	2:	IF TIME() - T_dimm_start >= tx THEN
			state := 3;
			tx := TIME();
			(* time to switch elapsed without switching if Q = 0 turn on output and start dimming at 1 *)
			IF NOT Q THEN
				Q := TRUE;
				t_on := tx;
				out := 1;
				dimm_up := TRUE;
			ELSE
				IF out =255 THEN dimm_up := FALSE; END_IF;
			END_IF;
		ELSIF in XOR edge THEN
			(* wait for edge to toggle output and stop all activity *)
			IF Q THEN
				Q := FALSE;
				state := 0;
			ELSE
				Q := TRUE;
				state := 3;
				IF out = 0 THEN out := 255; END_IF
				IF out = 255 THEN dimm_up := FALSE; END_IF;
				tx := TIME();
				t_on := tx;
			END_IF;
		END_IF;

	(* state 3 entered dimming phase *)
	3:	IF in AND r_edge THEN
			(* generate ramp *)
			tx := TIME();
			IF tx >= last_step + T_dimm / 255 THEN
				last_step := tx;
				IF dimm_up AND out < 255 THEN
					out := out + 1;
					IF out = 255 THEN
						dimm_up := FALSE;
						state := 0;
					END_IF;
				ELSIF NOT dimm_up AND out > 0 THEN
					out := out -1;
					IF out = 0 THEN
						Q := FALSE;
						state := 0;
						dimm_up := TRUE;
					 END_IF;
				 END_IF;
			END_IF;
		ELSE
			dimm_up := NOT dimm_up;
			state := 0;
		END_IF;

	END_CASE;
	(* check for max t_on time and reset output if too long *)
	IF Q AND t_on_max > T#0s AND TIME() - t_on_max >= T_on THEN Q := 0; END_IF;

	(* check for reconfig and set R_edge to high for rising edge sensitivity *)
	IF TIME() - T_reconfig >= tx THEN R_edge := NOT in; END_IF;

	(* set edge to follow in for next edge detection *)
	edge := in;
END_IF;
END_FUNCTION_BLOCK

(* POU engineering/signal generators/rmp_B, ST *)
FUNCTION_BLOCK rmp_B
VAR_INPUT
	SET : BOOL := FALSE;
	PT : TIME;
	EN : BOOL := TRUE;
	UD : BOOL := TRUE;
	RST : BOOL := FALSE;
END_VAR
VAR_OUTPUT
	Out : BYTE := 0;
	busy: BOOL;
END_VAR
VAR
	last_step : TIME := T#0ms;
	step: TIME := T#0ms;
	now : TIME;
END_VAR

(*
	version 1.1	5 oct 2006
	programmer 	oscat
	tested BY		oscat

this ramp generator generates a byte wide ramp with 255 steps
the generator has an asynchronous set and reset
the ramp is controlled by PT which is the total ramp time for a full sweep from 0..255
an UD input controlls the direction Up or Down and the E input enables the ramp generation
a busy output indicates that the ramp is running, busy false means output is stable.

*)
IF en  THEN
	(* generate ramp *)
	now := TIME();
	IF now >= last_step + pt / 255 THEN
		last_step := now;
		IF UD AND out < 255 THEN out := out + 1; END_IF;
		IF NOT ud AND out > 0 THEN out := out -1; END_IF;
	END_IF;
END_IF;

(* check for asynchronous set or reset *)
IF set  THEN out := 255; END_IF;
IF rst THEN out := 0; END_IF;

(* checks for outputs stable and reset or set busy flag *)
IF out = 0 OR out = 255 THEN busy := FALSE; ELSE busy := TRUE; END_IF;
END_FUNCTION_BLOCK

(* POU String/exec, ST *)
FUNCTION exec : STRING
VAR_INPUT
	str : STRING;
END_VAR
VAR
	pos: INT;
	R1: REAL;
	R2: REAL;
	operator: STRING;
END_VAR

(*
version 1.0	6 oct 2006
programmer 	hugo
tested by		tobias

exec executes a mathematical term and returns the result as a string
the term can only be a simple term without brackets and only one operator
allowed operastors are: (+, -, *, /, ^, sqrt, sin, cos, tan).

*)
(* extract both numbers and operator *)
exec := uppercase(trim(str));
pos := findB_nonum(exec);
IF pos > 1 THEN R1 := STRING_TO_REAL(exec); END_IF;
R2 := STRING_TO_REAL(RIGHT(exec,LEN(exec)-pos));
exec := LEFT(exec,pos);
pos := findB_Num(exec);
operator := RIGHT(exec,LEN(exec) - pos);
IF operator = '' AND LEN(str) = 0 THEN
	exec := '';
	RETURN;
ELSIF operator = '' THEN
	exec := str;
	RETURN;
END_IF;
IF operator = '^' THEN
	exec := REAL_TO_STRING(EXPT(R1, R2));
ELSIF operator = 'SQRT' THEN
	exec := REAL_TO_STRING(SQRT(R2));
ELSIF operator = 'SIN' THEN
	exec := REAL_TO_STRING(SIN(r2));
ELSIF operator = 'cos' THEN
	exec := REAL_TO_STRING(COS(r2));
ELSIF operator = 'TAN' THEN
	exec := REAL_TO_STRING(TAN(R2));
ELSIF operator = '*' THEN
	exec := REAL_TO_STRING(R1 * R2);
ELSIF operator = '/' THEN
	exec := REAL_TO_STRING(R1 / R2);
ELSIF operator = '+' THEN
	exec := REAL_TO_STRING(r1 + r2);
ELSIF operator = '-' THEN
	exec := REAL_TO_STRING(r1 - r2);
ELSE
	exec := 'ERROR';
END_IF;
END_FUNCTION

(* POU String/uppercase, ST *)
FUNCTION uppercase : STRING
VAR_INPUT
	str : STRING;
END_VAR
VAR
	PT : POINTER TO BYTE;
	pos: INT;
END_VAR

(*
version 1.0	6 oct 2006
programmer 	hugo
tested by		tobias

uppercase returns str while all letters a..z are converted to uppercase

*)
PT := ADR(uppercase);
uppercase := str;
FOR pos := 1 TO LEN(str) DO
	IF PT^ > 96 AND PT^ < 123 THEN PT^ := PT^ - 32; END_IF;
	PT := PT + 1;
END_FOR;
END_FUNCTION

(* POU String/trim, ST *)
FUNCTION trim : STRING
VAR_INPUT
	str : STRING;
END_VAR
VAR
	pos: INT;
END_VAR

(*
version 1.0	6 oct 2006
programmer 	hugo
tested by		tobias

the function deletes all blaks within a string.

*)
trim := str;
REPEAT
	pos := FIND(trim,' ');
	trim := REPLACE(trim,'',1,pos);
UNTIL pos = 0	END_REPEAT;
END_FUNCTION

(* POU String/findB_nonum, ST *)
FUNCTION findB_nonum : INT
VAR_INPUT
	str : STRING;
END_VAR
VAR
	pos: INT;
	pt : POINTER TO BYTE;
END_VAR

(*
version 1.0	6 oct 2006
programmer 	hugo
tested by		tobias

findB_noNum searches str backwards and returns the last position which is not a number.
a number is characterized by a letter "0..9" or "."

*)
pt := ADR(str) + LEN(str) - 1;
findB_nonum := 0;
FOR pos := LEN(str) TO 1 BY -1 DO;
	IF NOT((PT^ > 47 AND PT^ < 58) OR PT^ = 46) THEN
		findB_nonum := pos;
		RETURN;
	END_IF;
	PT := PT - 1;
END_FOR;
END_FUNCTION

(* POU String/findB_Num, ST *)
FUNCTION findB_Num : INT
VAR_INPUT
	str : STRING;
END_VAR
VAR
	pos: INT;
	pt : POINTER TO BYTE;
END_VAR

(*
version 1.0	6 oct 2006
programmer 	hugo
tested by		tobias

findB_Num searches str backward and returns the last position of a number
a number is characterized by a letter "0..9" or "."

*)
pt := ADR(str) + LEN(str) - 1;
findB_Num := 0;
FOR pos := LEN(str) TO 1 BY -1 DO;
	IF (PT^ > 47 AND PT^ < 58) OR PT^ = 46 THEN
		findB_Num := pos;
		RETURN;
	END_IF;
	PT := PT - 1;
END_FOR;
END_FUNCTION

(* POU mathematical/functions/F_lin, ST *)
FUNCTION F_lin : REAL
VAR_INPUT
	X : REAL;
	A : REAL;
	B : REAL;
END_VAR
VAR
END_VAR

(*
version 1.0	1 sep 2006
programmer 	hugo
tested by		tobias

this function calculates the linear equation f_lin = a*x + b

*)
F_lin := A * X + B;
END_FUNCTION

(* POU mathematical/functions/F_power, ST *)
FUNCTION F_power : REAL
VAR_INPUT
	a : REAL;
	x : REAL;
	n : REAL;
END_VAR
VAR
END_VAR

(*
version 1.0	1 sep 2006
programmer 	hugo
tested by		tobias

this function calculates the power equation f_power = a*x^n

*)
f_power := a * EXPT(X,N);
END_FUNCTION

(* POU mathematical/functions/F_quad, ST *)
FUNCTION F_quad : REAL
VAR_INPUT
	X : REAL;
	A : REAL;
	B : REAL;
	C : REAL;
END_VAR
VAR
END_VAR

(*
version 1.0	1 sep 2006
programmer 	hugo
tested by		tobias

this function calculates the quadratic equation f_lin = a*x + b

*)
F_quad := a * X * X + B * X + C;
END_FUNCTION

(* POU engineering/conversion/F_to_C, ST *)
FUNCTION F_to_C : REAL
VAR_INPUT
	fahrenheit : REAL;
END_VAR
VAR
END_VAR

(*
version 1.0	4 aug 2006
programmer 	hugo
tested BY		tobias

this FUNCTION converts fahrenheit TO celsius

executioin TIME on wago 750-841 = 15us
*)
F_to_C := (fahrenheit -32) / 1.8;
END_FUNCTION

(* POU engineering/conversion/F_to_PT, ST *)
FUNCTION F_to_PT : TIME
VAR_INPUT
	F : REAL;
END_VAR
VAR
END_VAR

(*
version 1.0	4 aug 2006
programmer 	hugo
tested by		tobias

this function converts frequency to periode time  
*)
F_to_PT := DWORD_TO_TIME(REAL_TO_DWORD(1/F*1000));
END_FUNCTION

(* POU mathematical/fact, ST *)
FUNCTION fact : INT
VAR_INPUT
	X : INT;
END_VAR
VAR
	i: INT;
END_VAR

(*
version 1.0	1 sep 2006
programmer 	hugo
tested by		tobias

this function calculates the factorial of x
this simple factorial only calculates factorials for inputs up to 7
if the input is negative or higher then 7 the output will be -1.

*)
IF x >= 0 AND x < 8 THEN
	fact := 1;
	i := 2;
	WHILE x < i DO
		fact := fact * i;
	END_WHILE;
ELSE fact := -1;
END_IF;
END_FUNCTION

(* POU Logic/FF edge triggered/FF_D2E, ST *)
FUNCTION_BLOCK FF_D2E
VAR_INPUT
	D0 : BOOL := 0;
	D1 : BOOL := 0;
	CLK : BOOL;
	RST : BOOL := 0;
END_VAR
VAR_OUTPUT
	Q0 : BOOL := 0;
	Q1 : BOOL := 0;
END_VAR
VAR
	edge : BOOL;
END_VAR

(*
version 1.0	4 aug 2006
programmer 	hugo
tested by		tobias

dual D-type flip flop with reset and rising clock trigger

executioin TIME on wago 750-841 = 6us
*)
IF rst THEN
	Q0 := FALSE;
	Q1 := FALSE;
ELSE
	IF clk AND NOT edge THEN
		Q0 := D0;
		Q1 := D1;
	END_IF;
END_IF;
edge := CLK;
END_FUNCTION_BLOCK

(* POU Logic/FF edge triggered/FF_D4E, ST *)
FUNCTION_BLOCK FF_D4E
VAR_INPUT
	D0 : BOOL := 0;
	D1 : BOOL := 0;
	D2 : BOOL := 0;
	D3 : BOOL := 0;
	CLK : BOOL;
	RST : BOOL := 0;
END_VAR
VAR_OUTPUT
	Q0 : BOOL := 0;
	Q1 : BOOL := 0;
	Q2 : BOOL := 0;
	Q3 : BOOL := 0;
END_VAR
VAR
	edge : BOOL;
END_VAR


(*
version 1.0	4 aug 2006
programmer 	hugo
tested by		tobias

quad D-type flip flop with reset and rising clock trigger

executioin TIME on wago 750-841 = 6us
*)
IF rst THEN
	Q0 := FALSE;
	Q1 := FALSE;
	Q2 := FALSE;
	Q3 := FALSE;
ELSE
	IF clk AND NOT edge THEN
		Q0 := D0;
		Q1 := D1;
		Q2 := D2;
		Q3 := D3;
	END_IF;
END_IF;
edge := CLK;
END_FUNCTION_BLOCK

(* POU Logic/FF edge triggered/FF_DRE, ST *)
FUNCTION_BLOCK FF_DRE
VAR_INPUT
	set : BOOL;
	D : BOOL;
	CLK : BOOL;
	RST : BOOL;
END_VAR
VAR_OUTPUT
	Q : BOOL := 0;
END_VAR
VAR
	edge : BOOL;
END_VAR


(*
version 1.0	4 aug 2006
programmer 	hugo
tested by		tobias

D-type flip flop with set, reset and rising clock trigger
executioin TIME on wago 750-841 = 8us
*)
IF rst THEN
	Q := FALSE;
ELSIF set AND NOT rst THEN
	Q := TRUE;
ELSE
	IF clk AND NOT edge THEN Q := D; END_IF;
END_IF;
edge := CLK;
END_FUNCTION_BLOCK

(* POU Logic/FF edge triggered/FF_JKE, ST *)
FUNCTION_BLOCK FF_JKE
VAR_INPUT
	SET : BOOL;
	J : BOOL;
	CLK : BOOL;
	K : BOOL;
	RST : BOOL;
END_VAR
VAR_OUTPUT
	Q : BOOL := 0;
END_VAR
VAR
	edge : BOOL;
END_VAR


(*
version 1.0	4 aug 2006
programmer 	hugo
tested by		tobias

JK-type flip flop with set, reset and rising clock trigger
set and reset are asynchron while the FF is rising edge triggered
J=0 and K=0 and CLK >>> no action
J=1 and K=0 and CLK >>> output = 1
J=0 and K=1 and CLK >>> output = 0
J=1 and K=1 and CLK >>> toggle output

executioin TIME on wago 750-841 = 8us
*)
IF rst THEN
	Q := FALSE;
ELSIF set AND NOT rst THEN
	Q := TRUE;
ELSE
	IF clk AND NOT edge THEN
		IF J AND NOT K THEN Q := TRUE;
		ELSIF K AND NOT J THEN Q := FALSE;
		ELSIF K AND J THEN Q:= NOT Q;
		END_IF;
	END_IF;
END_IF;
edge := CLK;
END_FUNCTION_BLOCK

(* POU Logic/memory/FIFO_16, ST *)
FUNCTION_BLOCK FIFO_16
VAR_INPUT
	Din : DWORD;
	WR : BOOL;
	E : BOOL;
	RST : BOOL;
END_VAR
VAR_OUTPUT
	Dout : DWORD := 0;
	empty : BOOL := TRUE;
	full : BOOL := FALSE;
END_VAR
VAR
	fifo : ARRAY[0..15] OF DWORD;
	NW : INT := 0;
	NR : INT := 0;
	top : INT := 15;
END_VAR

(*
	version 1.0	4 aug 2006
	programmer 	hugo
	tested by		tobias

16 Dword FIFO memory
*)
IF rst THEN
	(* asynchronous reset for the fifo *)
	NW := 0;
	NR := 0;
	Dout := 0;
	empty := TRUE;
	full := FALSE;
ELSIF WR AND E AND NOT full THEN
	(* write action *)
	fifo[NW] := Din;
	IF NW = top THEN NW := 0; ELSE NW := NW + 1; END_IF
	IF NW = NR THEN full := TRUE; END_IF
	empty := FALSE;
ELSIF NOT WR AND E AND NOT empty THEN
	(* read from stack *)
	Dout := fifo[NR];
	IF NR = top THEN NR := 0; ELSE NR := NR + 1; END_IF;
	IF NR = NW THEN empty := TRUE; END_IF;
	full := FALSE;
END_IF;
END_FUNCTION_BLOCK

(* POU Logic/memory/FIFO_32, ST *)
FUNCTION_BLOCK FIFO_32
VAR_INPUT
	Din : DWORD;
	WR : BOOL;
	E : BOOL;
	RST : BOOL;
END_VAR
VAR_OUTPUT
	Dout : DWORD := 0;
	empty : BOOL := TRUE;
	full : BOOL := FALSE;
END_VAR
VAR
	fifo : ARRAY[0..31] OF DWORD;
	NW : INT := 0;
	NR : INT := 0;
	top : INT := 31;
END_VAR

(*
	version 1.0	4 aug 2006
	programmer 	hugo
	tested by		tobias

32 Dword FIFO memory
*)
IF rst THEN
	(* asynchronous reset for the fifo *)
	NW := 0;
	NR := 0;
	Dout := 0;
	empty := TRUE;
	full := FALSE;
ELSIF WR AND E AND NOT full THEN
	(* write action *)
	fifo[NW] := Din;
	IF NW = top THEN NW := 0; ELSE NW := NW + 1; END_IF
	IF NW = NR THEN full := TRUE; END_IF
	empty := FALSE;
ELSIF NOT WR AND E AND NOT empty THEN
	(* read from stack *)
	Dout := fifo[NR];
	IF NR = top THEN NR := 0; ELSE NR := NR + 1; END_IF;
	IF NR = NW THEN empty := TRUE; END_IF;
	full := FALSE;
END_IF;
END_FUNCTION_BLOCK

(* POU String/find_nonum, ST *)
FUNCTION find_nonum : INT
VAR_INPUT
	str : STRING;
END_VAR
VAR
	pos: INT;
	pt : POINTER TO BYTE;
END_VAR

(*
version 1.0	6 oct 2006
programmer 	hugo
tested by		tobias

find_noNum searches str and returns the first position which is not a number.
a number is characterized by a letter "0..9" or "."

*)
pt := ADR(str);
find_nonum := 0;
FOR pos := 1 TO LEN(str) DO;
	IF NOT((PT^ > 47 AND PT^ < 58) OR PT^ = 46) THEN
		find_nonum := pos;
		RETURN;
	END_IF;
	PT := PT + 1;
END_FOR;
END_FUNCTION

(* POU String/find_Num, ST *)
FUNCTION find_Num : INT
VAR_INPUT
	str : STRING;
END_VAR
VAR
	pos: INT;
	pt : POINTER TO BYTE;
END_VAR

(*
version 1.0	6 oct 2006
programmer 	hugo
tested by		tobias

find_Num searches str and returns the starting position of a number
a number is characterized by a letter "0..9" or "."

*)
pt := ADR(str);
find_Num := 0;
FOR pos := 1 TO LEN(str) DO;
	IF (PT^ > 47 AND PT^ < 58) OR PT^ = 46 THEN
		find_Num := pos;
		RETURN;
	END_IF;
	PT := PT + 1;
END_FOR;
END_FUNCTION

(* POU String/FindB, ST *)
FUNCTION FindB : INT
VAR_INPUT
	str1 : STRING;
	str2 : STRING;
END_VAR
VAR
	pos: INT;
	size: INT;
	length: INT;
END_VAR

(*
version 1.0	6 oct 2006
programmer 	hugo
tested by		tobias

the function find searches an str1 for the presence of str2 and returns the first position of str1 of the last presence in instring.
the function is similar to find except it searches from the right to left.
 a 0 is returned if the string is not found.

*)
size := LEN(str1);
length := LEN(str2);
FOR pos := size TO 1 BY -1 DO
	IF MID(str1,length,pos) = str2 THEN
		FindB := pos;
		RETURN;
	END_IF;
END_FOR;
END_FUNCTION

(* POU mathematical/fract, ST *)
FUNCTION fract : REAL
VAR_INPUT
	input : REAL;
END_VAR
VAR
END_VAR
VAR
END_VAR

(*
version 1.0	4 aug 2006
programmer 	hugo
tested by		tobias

this function returns the fraction of a real number
fract(3.14) = 0.14

execution time on wago 750 - 841 =  17  us
*)
fract := input - TRUNC(input);
END_FUNCTION

(* POU mathematical/functions/FT_avg, ST *)
FUNCTION_BLOCK FT_avg
VAR_INPUT
	in : REAL;
	N : INT;
	rst : BOOL;
END_VAR
VAR_OUTPUT
	avg : REAL;
END_VAR
VAR
	buff : delay;
END_VAR

(*
version 1.0	1 oct 2006
programmer 	hugo
tested by		tobias

this function calculates the average over n samples from a sequential input
the input values are shifted into an N deep buffer and the avg of this buffer is diplayed at anytime on the output.
a rst will clear the buffer at any time.

*)
IF N > 32 THEN N:= 32; END_IF;
buff.N := N;
IF rst THEN
	buff(rst := TRUE);
	buff.rst := FALSE;
	avg := 0;
ELSE
	buff(in := in);
	avg := avg + (in - buff.out)/N;
END_IF;
END_FUNCTION_BLOCK

(* POU mathematical/functions/FT_deriv, ST *)
FUNCTION_BLOCK FT_deriv
VAR_INPUT
	in : REAL;
	K : REAL;
	run : BOOL := 1;
END_VAR
VAR_OUTPUT
	out : REAL;
END_VAR
VAR
	old: REAL;
	tx: TIME;
	last: TIME;
END_VAR


(*
version 1.0	1 oct 2006
programmer 	hugo
tested by		tobias

FT_deriv calculated the derivate over the signal "in" with Faktor "K".
a run input enables or stops the calculation, if left unconnected its true and therfore the calculation is executed.


*)
tx := TIME() - last;
IF run THEN
	out := (in - old) / TIME_TO_REAL(tx) * 1000 * K;
ELSE
	out := 0;
END_IF;
old := in;
last := tx + last;
END_FUNCTION_BLOCK

(* POU mathematical/functions/FT_INT, ST *)
FUNCTION_BLOCK FT_INT
VAR_INPUT
	in : REAL;
	K : REAL;
	run : BOOL := 1;
	rst: BOOL;
	out_min : REAL := -1000;
	out_max : REAL := 1000;
END_VAR
VAR_OUTPUT
	Out : REAL;
	ET: TIME;
END_VAR
VAR
	last: TIME;
	in_last : REAL;
END_VAR


(*
version 1.1	13 dec 2006
programmer 	hugo
tested by		tobias

FT_int is an integrator with input IN and factor K
integration is only done while run = true, if run is false integration is stopped and the out remains at the last value.
if run is left unconnected, run is considered true by the function block.
the output ET will display the total integration time from last reset.
a rst input will reset output and the timer ET to 0.
the out_min and out_max values can be set to ,imit the output value range. 
out _min is preset to -1000 and out_max is preset to 1000.

 
*)
IF rst THEN
	out := 0;
	ET := t#0s;
ELSIF run THEN
	out := out + (in + in_last)/2 * TIME_TO_DINT(TIME()-last) * K / 1000;
	IF out < out_min THEN out := out_min; ELSIF out > out_max THEN out := out_max; END_IF;
	et := et + TIME() - last;
END_IF;
last := TIME();
in_last := in;
(*
hm 13.12.2006	rev 1.1
changed to "trapezregel" which increases accuracy
before out := out + in * time new: out := out + (in + in_last) / 2 * time

*)
END_FUNCTION_BLOCK

(* POU mathematical/functions/FT_min_max, ST *)
FUNCTION_BLOCK FT_min_max
VAR_INPUT
	in : REAL;
	rst : BOOL;
END_VAR
VAR_OUTPUT
	mx : REAL;
	mn : REAL;
END_VAR
VAR
	init: BOOL;
END_VAR

(*
version 1.0	1 sep 2006
programmer 	hugo
tested by		tobias

this function block stores the min and max value of an input signal.
when rst is true the mn and mx outputs are set to the in value.
when a rst is never active the function autoresets to the in value at startup.
since the input might not be present at first cycle the mn and mx are set during second cycle.

*)
IF rst OR NOT init THEN
	mn := in;
	mx := in;
	init := 1;
ELSIF in < mn THEN mn := in;
ELSIF in > mx THEN mx := in;
END_IF;
END_FUNCTION_BLOCK

(* POU engineering/FT_PID, ST *)
FUNCTION_BLOCK FT_PID
VAR_INPUT
	actual, set_point, offset, manual_in : REAL;
	Manual : BOOL;
	rst : BOOL := FALSE;
END_VAR
VAR_INPUT
	KP, TN, TV, limit_L, limit_H : REAL;
END_VAR
VAR_OUTPUT
	Y : REAL;
	LIM, overflow : BOOL;
END_VAR
VAR
	integ : FT_INT;
	deriv : FT_deriv;
	diff: REAL;
END_VAR

(*
version 1.1	25 dec 2006
programmer 	hugo
tested by		tobias

FT_PID is a pid controller with manual functionality.
The PID controller works according to the fomula Y = KP * ( e + 1/TN * INTEG(e) + TV *DERIV(e)) + offset, while e = set_point - actual.
a rst will reset all internal data, while a switch to manual will cause the controller to follow the function Y = manual_in + offset.
limit_h and Limit_l set the possible output range of Y.
the output flags lim will signal that the output limits are active and overflow will signal that the integrator has reached the max or min limit.  

since rev 1.1 the "trapezregel is used for more accuracy. 
*)
IF rst OR KP = 0 THEN
	y := offset;
	integ(rst := 1);
	integ.rst := 0;
ELSIF manual THEN
	Y := manual_in + offset;
	integ(rst := 1);
	integ.rst := 0;
ELSE
	(* calcualtion of the actual PID values *)
	diff := set_point - actual;

	(* integrator is only called if TN > 0 othewrwise it is disabled *)
	IF TN > 0 THEN integ(in := diff, K := 1/TN, out_min := (limit_L - offset) / KP, out_max := (limit_H - offset) / KP); END_IF;
	deriv(in := diff, K := TV);

	(* check if integrator has reached the allowed limits and set overflow if necessary *)
	IF integ.Out >= (limit_H - offset) / KP THEN
		Y := limit_H;
		overflow := TRUE;
	ELSIF integ.Out <= (limit_L - offset) / KP THEN
		Y := limit_L;
		overflow := TRUE;
	ELSE
		Y := KP * (integ.Out + deriv.out + diff) + offset;
		overflow := FALSE;
	END_IF;

	(* this portion limits the output to limit_H and limit_L and set the lim flag if limits are exceeded *)
	IF Y > limit_H THEN
		Y := limit_H;
		Lim := TRUE;
	ELSIF Y < limit_L THEN
		Y := limit_L;
		lim := TRUE;
	ELSE
		lim := FALSE;
	END_IF;
END_IF;
END_FUNCTION_BLOCK

(* POU mathematical/functions/FT_PT1, ST *)
FUNCTION_BLOCK FT_PT1
VAR_INPUT
	in : REAL;
	T : TIME;
END_VAR
VAR_OUTPUT
	out : REAL;
END_VAR
VAR
	last : TIME;
END_VAR

(*
version 1.0	1 oct 2006
programmer 	hugo
tested by		tobias

FT_PT1 is an low pass filter with a programmable time T.
 
*)
IF T = t#0s THEN
	out := in;
ELSE
	out := out + (in - out) * TIME_TO_REAL(TIME() - last) / TIME_TO_REAL(T);
END_IF;
last := TIME();
END_FUNCTION_BLOCK

(* POU Logic/generators/gen_bit, ST *)
FUNCTION_BLOCK gen_bit
VAR_INPUT
	in0 : DWORD;
	in1 : DWORD;
	in2 : DWORD;
	in3 : DWORD;
	clk : BOOL := 0;
	steps : INT;
	rep : INT := 0;
	rst : BOOL := 0;
END_VAR
VAR_OUTPUT
	Q0 :BOOL := 0;
	Q1 :BOOL := 0;
	Q2 :BOOL := 0;
	Q3 :BOOL := 0;
	cnt : INT := 0;
	run : BOOL := 0;
END_VAR
VAR
	r0: DWORD;
	r1: DWORD;
	r2: DWORD;
	r3: DWORD;
	rx : INT := 1;
END_VAR

(*
version 1.0	4 aug 2006
programmer 	hugo
tested by		tobias

clk_prg uses the internal sps time to generate a clock with programmable period time.
the period time is defined for 1ms .. 65s
the first cycle after start is a clk pulse and then depending on the programmed period time a delay.
every pulse is only valid for one cycle so that a edge trigger is not necessary
clk_prg depending on the accuracy of the system clock.

*)
(* check if number of runs is finished or rep = 0 which means continuous *)

IF clk AND NOT rst THEN
	IF (rep = 0) OR (rx <= rep) THEN run := TRUE; ELSE run := FALSE; END_IF;
	IF run THEN
		(* check for step counter reached and reset to 0 if cnt = steps *)
		IF cnt = steps THEN
			cnt := 0;
		END_IF;

		(* when cnt = 0 then reload the inputs into the registers *)
		IF cnt = 0 THEN
			r0 := in0;
			r1 := in1;
			r2 := in2;
			r3 := in3;
		END_IF;

		(* when cnt < steps, shift the lowest bits to the outputs *)
		IF (cnt < steps) THEN
			Q0 := r0.0;
			Q1 := r1.0;
			Q2 := r2.0;
			Q3 := r3.0;
			r0 := SHR(r0,1);
			r1 := SHR(r1,1);
			r2 := SHR(r2,1);
			r3 := SHR(r3,1);
		END_IF;

		(* increment the step counter *)
		cnt := cnt +1;
		IF (cnt = steps) AND (rep <> 0) THEN rx := rx +1; END_IF;
		IF (rx > rep) AND (rep <> 0) THEN run := FALSE; END_IF;
	END_IF;
ELSE
	IF rst THEN
		Q0 := FALSE;
		Q1 := FALSE;
		Q2 := FALSE;
		Q3 := FALSE;
		r0 := 0;
		r1 := 0;
		r2 := 0;
		r3 := 0;
		cnt := 0;
		run := FALSE;
		rx := 1;
	END_IF;
END_IF;
END_FUNCTION_BLOCK

(* POU Logic/generators/gen_SQ, ST *)
FUNCTION_BLOCK gen_SQ
VAR_INPUT
	PT : TIME := T#0ms;
END_VAR
VAR_OUTPUT
	Q : BOOL := 0;
END_VAR
VAR
	pti : TIME := t#0ms;
	run: BOOL := FALSE;
	next_edge: TIME := t#0ms;
	overflow: BOOL := 0;
END_VAR

(*
version 1.0	4 aug 2006
programmer 	hugo
tested by		tobias

gen_sq generates square wave signal with programmable period time.
the period time is defined for 10ms .. 65s
if the period time is set to less then 10ms the min perid is 10ms.

*)
IF NOT run THEN
	next_edge := TIME();
	run := TRUE;
	IF pt < T#10ms THEN PTI := T#5ms; ELSE pti := pt/2; END_IF;
END_IF;
IF (TIME() >= next_edge) AND NOT overflow THEN
	Q := NOT Q;
	IF next_edge + pti < next_edge THEN
		(* time() will overflow every 50 days *)
		overflow := TRUE;
	END_IF;
	next_edge := next_edge + pti;
ELSE
	(* wait till time() has an overflow and reset overflow *)
	IF TIME() <= next_edge THEN overflow := FALSE; END_IF;
END_IF;
END_FUNCTION_BLOCK

(* POU Time&Date/hour_to_time, ST *)
FUNCTION hour_to_time : TIME
VAR_INPUT
	input : REAL;
END_VAR
VAR
END_VAR

(*
version 1.0	4 aug 2006
programmer 	hugo
tested by		tobias

converts an amount of hours in real to time
execution TIME on wago 750-841 =  17us
*)
hour_to_time := DWORD_TO_TIME(REAL_TO_DWORD(input * 3600000));
END_FUNCTION

(* POU Time&Date/hour_to_tod, ST *)
FUNCTION hour_to_tod : TOD
VAR_INPUT
	input : REAL;
END_VAR
VAR
END_VAR

(*
version 1.0	4 aug 2006
programmer 	hugo
tested by		tobias

converts an amount of hours in real to time of day 
execution time on wago 750-841 =  17us 
*)
hour_to_tod := DWORD_TO_TOD(REAL_TO_DWORD(input * 3600000));
END_FUNCTION

(* POU engineering/measurements/hyst_1, ST *)
FUNCTION_BLOCK hyst_1
VAR_INPUT
	In : REAL;
	high : REAL;
	low : REAL;
END_VAR
VAR_OUTPUT
	Q : BOOL := 0;
	win : BOOL := 0;
END_VAR
VAR
END_VAR

(*
	version 1.0	4 aug 2006
	programmer 	hugo
	tested BY		tobias

this hysteresis function switches the output high if the input signal reaches obove high and will switch to low when the input falls back below low value.
a separate output mid is set if the input stays between low and high value.

*)
IF Q THEN
	IF in < low THEN q := FALSE; END_IF;
ELSE
	IF in > high THEN q := TRUE; END_IF;
END_IF;
win := in > low AND in < high;
END_FUNCTION_BLOCK

(* POU engineering/measurements/hyst_2, ST *)
FUNCTION_BLOCK hyst_2
VAR_INPUT
	In : REAL;
	val : REAL;
	hys : REAL;
END_VAR
VAR_OUTPUT
	Q : BOOL := 0;
	win: BOOL;
END_VAR
VAR
	X : REAL;
END_VAR


(*
	version 1.0	4 aug 2006
	programmer 	oscat
	tested BY		tobias

this hysteresis function switches the output high if the input signal reaches obove val + hys/2 and will switch to low when the input falls back below val - hys/2 value.
a separate output mid is set if the input stays between low and high value.

*)
X := hys / 2;
IF Q THEN
	IF in < val - x THEN q := FALSE; END_IF;
ELSE
	IF in > val + x THEN q := TRUE; END_IF;
END_IF;
win := in > val - x AND in < val + x;
END_FUNCTION_BLOCK

(* POU engineering/measurements/inc_dec, ST *)
FUNCTION_BLOCK inc_dec
VAR_INPUT
	CHa : BOOL;
	CHb : BOOL;
	RST : BOOL := 0;
END_VAR
VAR_OUTPUT
	dir : BOOL;
	cnt : INT;
END_VAR
VAR
	edge : BOOL := 0;
	edgea : BOOL := 0;
	clk: BOOL;
	clka: BOOL;
	clkb: BOOL;
	edgeb: BOOL;
	axb: BOOL;
END_VAR

(*
	version 1.0	4 aug 2006
	programmer 	oscat
	tested BY		oscat

incremental decoder with quadruple accuracy.
2 pulses for each channel are created for each directional pulse.
*)
axb := cha XOR chb;

(* create pulses for channel a *)
clka := cha XOR edgea;
edgea := cha;

clkb := chb XOR edgeb;
edgeb := chb;

(* create pulses for both channels *)
clk := clka OR clkb;

(* set the direction output *)
IF axb AND clka THEN dir := TRUE; END_IF;
IF axb AND clkb THEN dir := FALSE; END_IF;

(* increment or decrement the counter *)
IF clk AND dir THEN cnt := cnt + 1; END_IF;
IF clk AND NOT dir THEN cnt := cnt -1; END_IF;

(* reset the counter if rst active *)
IF rst THEN cnt := 0; END_IF;
END_FUNCTION_BLOCK

(* POU Time&Date/leap_of_Date, ST *)
FUNCTION leap_of_Date : BOOL
VAR_INPUT
	idate : DATE;
END_VAR
VAR
END_VAR

(*
version 1.1	2 oct 2006
programmer 	hugo
tested by		tobias


leap_year is true if the tested year is a leap year  
execution time on wago 750-841 =  30 us   
*)
leap_of_Date := leap_year(year(idate));


(* change history

2.10.2006		changes to rev 1.1
the function now calls leap_year to accomodate further accuracy.
the function now works for any year from 1970 to 2100

*)
END_FUNCTION

(* POU Time&Date/leap_year, ST *)
FUNCTION leap_year : BOOL
VAR_INPUT
	yr : INT;
END_VAR
VAR
END_VAR

(*
version 1.1	2 oct 2006
programmer 	hugo
tested by		tobias


leap_year is true if the tested year is a leap year  
execution time on wago 750-841 =  12 us    
*)
IF yr MOD 400 = 0 THEN leap_year := TRUE;
ELSIF yr MOD 100 = 0 THEN leap_year := FALSE;
ELSIF yr MOD 4 =0 THEN leap_year := TRUE;
ELSE leap_year := FALSE;
END_IF;


(* change history

2.10.2006		changes to rev 1.1
the function now works for any year from 1970 up to 2100

*)
END_FUNCTION

(* POU Building/HLK/legionella, CFC *)
FUNCTION_BLOCK legionella
VAR_INPUT
	manual : BOOL;
	temp_boiler : REAL;
	temp_return : REAL;
	DT_in: DT;
	rst : BOOL;
END_VAR
VAR_INPUT CONSTANT
	T_start: TOD := tod#03:00:00;
	day : INT := 7;
	temp_set : REAL := 70;
	temp_offset : REAL := 10;
	temp_hys : REAL := 5;
	t_max_heat: TIME := t#10m;
	t_max_ret : TIME := t#10m;
	tp_0: TIME := t#5m;
	tp_1: TIME := t#5m;
	tp_2: TIME := t#5m;
	tp_3: TIME := t#5m;
	tp_4: TIME := t#5m;
	tp_5: TIME := t#5m;
	tp_6: TIME := t#5m;
	tp_7: TIME := t#5m;
END_VAR
VAR_OUTPUT
	Heat : BOOL;
	pump : BOOL;
	error : BOOL;
	valve0 : BOOL;
	valve1 : BOOL;
	valve2 : BOOL;
	valve3 : BOOL;
	valve4 : BOOL;
	valve5 : BOOL;
	valve6 : BOOL;
	valve7 : BOOL;
	run: BOOL;
END_VAR
VAR
	X1: timer_1;
	x2: sequence_8;
	x3: hyst_1;
	x4: hyst_1;
END_VAR

(*
version 1.0	10. Dec 2006
programmer 	oscat
tested by		hans

